LIN {X -0.036,Y -601.709,Z 354.126,A 0.000,B 0.000,C 90.000,E1 238.663} C_DIS
LIN {X -0.086,Y -595.770,Z 354.117,A 0.000,B 0.000,C 90.000,E1 237.089} C_DIS
LIN {X 0.073,Y -585.449,Z 354.101,A 0.000,B 0.000,C 90.000,E1 234.149} C_DIS
LIN {X -0.004,Y -581.907,Z 354.095,A 0.000,B 0.000,C 90.000,E1 233.084} C_DIS
LIN {X -0.070,Y -577.067,Z 354.087,A 0.000,B 0.000,C 90.000,E1 231.743} C_DIS
LIN {X 0.016,Y -567.476,Z 354.072,A 0.000,B 0.000,C 90.000,E1 229.013} C_DIS
LIN {X -0.240,Y -562.093,Z 354.063,A 0.000,B 0.000,C 90.000,E1 227.391} C_DIS
LIN {X -0.222,Y -556.673,Z 354.054,A 0.000,B 0.000,C 90.000,E1 225.729} C_DIS
LIN {X -0.289,Y -550.328,Z 354.043,A 0.000,B 0.000,C 90.000,E1 223.785} C_DIS
LIN {X -0.119,Y -544.951,Z 354.034,A 0.000,B 0.000,C 90.000,E1 222.081} C_DIS
LIN {X -0.053,Y -538.814,Z 354.023,A 0.000,B 0.000,C 90.000,E1 220.092} C_DIS
LIN {X -0.082,Y -532.771,Z 354.012,A 0.000,B 0.000,C 90.000,E1 218.096} C_DIS
LIN {X -0.221,Y -525.363,Z 353.997,A 0.000,B 0.000,C 90.000,E1 215.518} C_DIS
LIN {X 0.006,Y -519.158,Z 353.984,A 0.000,B 0.000,C 90.000,E1 213.166} C_DIS
LIN {X -0.145,Y -512.839,Z 353.970,A 0.000,B 0.000,C 90.000,E1 210.541} C_DIS
LIN {X 0.158,Y -508.202,Z 353.958,A 0.000,B 0.000,C 90.000,E1 208.437} C_DIS
LIN {X 0.158,Y -504.896,Z 353.950,A 0.000,B 0.000,C 90.000,E1 206.950} C_DIS
LIN {X 0.090,Y -501.709,Z 353.942,A 0.000,B 0.000,C 90.000,E1 205.463} C_DIS
LIN {X 0.192,Y -498.425,Z 353.933,A 0.000,B 0.000,C 90.000,E1 203.951} C_DIS
LIN {X 0.088,Y -494.313,Z 353.923,A 0.000,B 0.000,C 90.000,E1 202.153} C_DIS
LIN {X -0.187,Y -491.537,Z 353.916,A 0.000,B 0.000,C 90.000,E1 200.972} C_DIS
LIN {X -0.168,Y -487.311,Z 353.906,A 0.000,B 0.000,C 90.000,E1 199.141} C_DIS
LIN {X -0.098,Y -481.349,Z 353.891,A 0.000,B 0.000,C 90.000,E1 196.370} C_DIS
LIN {X 0.032,Y -476.989,Z 353.879,A 0.000,B 0.000,C 90.000,E1 194.189} C_DIS
LIN {X 0.059,Y -472.858,Z 353.867,A 0.000,B 0.000,C 90.000,E1 192.007} C_DIS
LIN {X -0.222,Y -468.764,Z 353.855,A 0.000,B 0.000,C 90.000,E1 189.849} C_DIS
LIN {X -0.227,Y -465.034,Z 353.842,A 0.000,B 0.000,C 90.000,E1 187.644} C_DIS
LIN {X -0.207,Y -461.052,Z 353.828,A 0.000,B 0.000,C 90.000,E1 185.106} C_DIS
LIN {X 0.195,Y -456.557,Z 353.809,A 0.000,B 0.000,C 90.000,E1 181.547} C_DIS
LIN {X -0.196,Y -452.824,Z 353.786,A 0.000,B 0.000,C 90.000,E1 177.421} C_DIS
LIN {X 0.187,Y -451.196,Z 353.768,A 0.000,B 0.000,C 90.000,E1 174.147} C_DIS
LIN {X 0.099,Y -450.799,Z 353.743,A 0.000,B 0.000,C 90.000,E1 169.634} C_DIS
LIN {X -0.141,Y -451.606,Z 353.726,A 0.000,B 0.000,C 90.000,E1 166.756} C_DIS
LIN {X 0.146,Y -454.119,Z 353.705,A 0.000,B 0.000,C 90.000,E1 162.851} C_DIS
LIN {X -0.169,Y -458.577,Z 353.682,A 0.000,B 0.000,C 90.000,E1 158.720} C_DIS
LIN {X 0.269,Y -464.355,Z 353.660,A 0.000,B 0.000,C 90.000,E1 154.845} C_DIS
LIN {X -0.128,Y -472.523,Z 353.638,A 0.000,B 0.000,C 90.000,E1 150.795} C_DIS
LIN {X 0.032,Y -482.123,Z 353.617,A 0.000,B 0.000,C 90.000,E1 147.041} C_DIS
LIN {X 0.035,Y -490.562,Z 353.602,A 0.000,B 0.000,C 90.000,E1 144.276} C_DIS
LIN {X -0.182,Y -496.597,Z 353.591,A 0.000,B 0.000,C 90.000,E1 142.477} C_DIS
LIN {X 0.047,Y -502.541,Z 353.581,A 0.000,B 0.000,C 90.000,E1 140.642} C_DIS
LIN {X -0.094,Y -506.324,Z 353.575,A 0.000,B 0.000,C 90.000,E1 139.461} C_DIS
LIN {X 0.147,Y -509.852,Z 353.568,A 0.000,B 0.000,C 90.000,E1 138.243} C_DIS
LIN {X -0.188,Y -512.384,Z 353.563,A 0.000,B 0.000,C 90.000,E1 137.391} C_DIS
LIN {X -0.238,Y -515.302,Z 353.557,A 0.000,B 0.000,C 90.000,E1 136.215} C_DIS
LIN {X 0.298,Y -516.581,Z 353.553,A 0.000,B 0.000,C 90.000,E1 135.567} C_DIS
LIN {X 0.024,Y -518.323,Z 353.548,A 0.000,B 0.000,C 90.000,E1 134.717} C_DIS
LIN {X 0.222,Y -519.271,Z 353.545,A 0.000,B 0.000,C 90.000,E1 134.109} C_DIS
LIN {X -0.014,Y -520.436,Z 353.540,A 0.000,B 0.000,C 90.000,E1 133.257} C_DIS
LIN {X 0.056,Y -521.438,Z 353.534,A 0.000,B 0.000,C 90.000,E1 132.081} C_DIS
LIN {X -0.154,Y -521.848,Z 353.529,A 0.000,B 0.000,C 90.000,E1 131.229} C_DIS
LIN {X 0.318,Y -521.762,Z 353.523,A 0.000,B 0.000,C 90.000,E1 130.011} C_DIS
LIN {X -0.233,Y -521.317,Z 353.518,A 0.000,B 0.000,C 90.000,E1 129.197} C_DIS
LIN {X -0.055,Y -520.533,Z 353.513,A 0.000,B 0.000,C 90.000,E1 128.302} C_DIS
LIN {X -0.209,Y -519.480,Z 353.508,A 0.000,B 0.000,C 90.000,E1 127.443} C_DIS
LIN {X -0.069,Y -517.552,Z 353.500,A 0.000,B 0.000,C 90.000,E1 125.964} C_DIS
LIN {X -0.253,Y -516.241,Z 353.495,A 0.000,B 0.000,C 90.000,E1 125.105} C_DIS
LIN {X -0.030,Y -514.817,Z 353.490,A 0.000,B 0.000,C 90.000,E1 124.199} C_DIS
LIN {X 0.092,Y -512.635,Z 353.483,A 0.000,B 0.000,C 90.000,E1 123.007} C_DIS
LIN {X -0.013,Y -510.853,Z 353.479,A 0.000,B 0.000,C 90.000,E1 122.133} C_DIS
LIN {X 0.199,Y -508.213,Z 353.472,A 0.000,B 0.000,C 90.000,E1 120.924} C_DIS
LIN {X 0.114,Y -505.440,Z 353.465,A 0.000,B 0.000,C 90.000,E1 119.745} C_DIS
LIN {X -0.005,Y -502.430,Z 353.459,A 0.000,B 0.000,C 90.000,E1 118.565} C_DIS
LIN {X -0.114,Y -498.474,Z 353.450,A 0.000,B 0.000,C 90.000,E1 117.078} C_DIS
LIN {X 0.146,Y -494.271,Z 353.442,A 0.000,B 0.000,C 90.000,E1 115.540} C_DIS
LIN {X 0.037,Y -491.575,Z 353.437,A 0.000,B 0.000,C 90.000,E1 114.643} C_DIS
LIN {X -0.058,Y -486.521,Z 353.429,A 0.000,B 0.000,C 90.000,E1 113.131} C_DIS
LIN {X 0.001,Y -482.302,Z 353.422,A 0.000,B 0.000,C 90.000,E1 111.897} C_DIS
LIN {X 0.004,Y -478.925,Z 353.417,A 0.000,B 0.000,C 90.000,E1 110.972} C_DIS
LIN {X 0.197,Y -475.980,Z 353.412,A 0.000,B 0.000,C 90.000,E1 110.174} C_DIS
LIN {X 0.128,Y -470.325,Z 353.404,A 0.000,B 0.000,C 90.000,E1 108.779} C_DIS
LIN {X 0.209,Y -465.075,Z 353.397,A 0.000,B 0.000,C 90.000,E1 107.511} C_DIS
LIN {X -0.253,Y -462.804,Z 353.395,A 0.000,B 0.000,C 90.000,E1 107.040} C_DIS
LIN {X 0.150,Y -462.797,Z 353.395,A 0.000,B 0.000,C 90.000,E1 106.985} C_DIS
LIN {X -0.040,Y -467.514,Z 353.383,A 0.000,B 0.000,C 90.000,E1 105.009} C_DIS
LIN {X -0.235,Y -468.097,Z 353.382,A 0.000,B 0.000,C 90.000,E1 104.717} C_DIS
LIN {X -0.096,Y -475.756,Z 353.357,A 0.000,B 0.000,C 90.000,E1 100.310} C_DIS
LIN {X 0.210,Y -476.285,Z 353.356,A 0.000,B 0.000,C 90.000,E1 99.962} C_DIS
LIN {X 0.158,Y -481.755,Z 353.331,A 0.000,B 0.000,C 90.000,E1 95.625} C_DIS
LIN {X 0.005,Y -482.163,Z 353.330,A 0.000,B 0.000,C 90.000,E1 95.334} C_DIS
LIN {X -0.066,Y -485.285,Z 353.306,A 0.000,B 0.000,C 90.000,E1 91.031} C_DIS
LIN {X -0.241,Y -485.538,Z 353.304,A 0.000,B 0.000,C 90.000,E1 90.745} C_DIS
LIN {X -0.034,Y -486.309,Z 353.282,A 0.000,B 0.000,C 90.000,E1 86.731} C_DIS
LIN {X 0.101,Y -486.319,Z 353.278,A 0.000,B 0.000,C 90.000,E1 86.102} C_DIS
LIN {X 0.174,Y -484.623,Z 353.253,A 0.000,B 0.000,C 90.000,E1 81.489} C_DIS
LIN {X 0.054,Y -480.552,Z 353.227,A 0.000,B 0.000,C 90.000,E1 76.881} C_DIS
LIN {X 0.150,Y -476.599,Z 353.212,A 0.000,B 0.000,C 90.000,E1 74.212} C_DIS
LIN {X 0.109,Y -476.610,Z 353.212,A 0.000,B 0.000,C 90.000,E1 74.212} C_DIS
LIN {X -0.055,Y -479.016,Z 353.210,A 0.000,B 0.000,C 90.000,E1 73.795} C_DIS
LIN {X 0.227,Y -482.346,Z 353.207,A 0.000,B 0.000,C 90.000,E1 73.142} C_DIS
LIN {X -0.158,Y -484.629,Z 353.204,A 0.000,B 0.000,C 90.000,E1 72.725} C_DIS
LIN {X -0.159,Y -486.303,Z 353.202,A 0.000,B 0.000,C 90.000,E1 72.417} C_DIS
LIN {X -0.046,Y -490.120,Z 353.198,A 0.000,B 0.000,C 90.000,E1 71.638} C_DIS
LIN {X 0.102,Y -493.632,Z 353.194,A 0.000,B 0.000,C 90.000,E1 70.859} C_DIS
LIN {X 0.240,Y -497.512,Z 353.189,A 0.000,B 0.000,C 90.000,E1 69.934} C_DIS
LIN {X -0.019,Y -500.472,Z 353.185,A 0.000,B 0.000,C 90.000,E1 69.209} C_DIS
LIN {X 0.195,Y -503.659,Z 353.180,A 0.000,B 0.000,C 90.000,E1 68.284} C_DIS
LIN {X -0.108,Y -505.682,Z 353.176,A 0.000,B 0.000,C 90.000,E1 67.720} C_DIS
LIN {X 0.267,Y -509.497,Z 353.170,A 0.000,B 0.000,C 90.000,E1 66.485} C_DIS
LIN {X -0.242,Y -513.111,Z 353.163,A 0.000,B 0.000,C 90.000,E1 65.357} C_DIS
LIN {X -0.020,Y -516.555,Z 353.156,A 0.000,B 0.000,C 90.000,E1 64.152} C_DIS
LIN {X -0.210,Y -519.929,Z 353.150,A 0.000,B 0.000,C 90.000,E1 62.999} C_DIS
LIN {X 0.031,Y -523.998,Z 353.142,A 0.000,B 0.000,C 90.000,E1 61.513} C_DIS
LIN {X -0.165,Y -528.825,Z 353.132,A 0.000,B 0.000,C 90.000,E1 59.793} C_DIS
LIN {X 0.065,Y -532.061,Z 353.126,A 0.000,B 0.000,C 90.000,E1 58.614} C_DIS
LIN {X 0.156,Y -536.027,Z 353.118,A 0.000,B 0.000,C 90.000,E1 57.168} C_DIS
LIN {X -0.137,Y -538.289,Z 353.113,A 0.000,B 0.000,C 90.000,E1 56.342} C_DIS
LIN {X 0.055,Y -541.226,Z 353.107,A 0.000,B 0.000,C 90.000,E1 55.182} C_DIS
LIN {X 0.126,Y -543.291,Z 353.102,A 0.000,B 0.000,C 90.000,E1 54.322} C_DIS
LIN {X -0.064,Y -545.864,Z 353.096,A 0.000,B 0.000,C 90.000,E1 53.210} C_DIS
LIN {X 0.101,Y -548.220,Z 353.089,A 0.000,B 0.000,C 90.000,E1 52.065} C_DIS
LIN {X -0.135,Y -550.313,Z 353.083,A 0.000,B 0.000,C 90.000,E1 50.964} C_DIS
LIN {X -0.046,Y -551.569,Z 353.078,A 0.000,B 0.000,C 90.000,E1 50.114} C_DIS
LIN {X 0.124,Y -552.673,Z 353.074,A 0.000,B 0.000,C 90.000,E1 49.256} C_DIS
LIN {X 0.187,Y -553.299,Z 353.071,A 0.000,B 0.000,C 90.000,E1 48.690} C_DIS
LIN {X -0.053,Y -553.923,Z 353.066,A 0.000,B 0.000,C 90.000,E1 47.877} C_DIS
LIN {X 0.110,Y -554.260,Z 353.060,A 0.000,B 0.000,C 90.000,E1 46.743} C_DIS
LIN {X -0.099,Y -553.911,Z 353.054,A 0.000,B 0.000,C 90.000,E1 45.648} C_DIS
LIN {X -0.013,Y -553.795,Z 353.051,A 0.000,B 0.000,C 90.000,E1 45.081} C_DIS
LIN {X -0.277,Y -553.292,Z 353.046,A 0.000,B 0.000,C 90.000,E1 44.271} C_DIS
LIN {X 0.232,Y -552.603,Z 353.041,A 0.000,B 0.000,C 90.000,E1 43.380} C_DIS
LIN {X 0.353,Y -551.766,Z 353.037,A 0.000,B 0.000,C 90.000,E1 42.528} C_DIS
LIN {X 0.103,Y -550.394,Z 353.030,A 0.000,B 0.000,C 90.000,E1 41.434} C_DIS
LIN {X -0.111,Y -549.020,Z 353.024,A 0.000,B 0.000,C 90.000,E1 40.334} C_DIS
LIN {X 0.106,Y -546.765,Z 353.015,A 0.000,B 0.000,C 90.000,E1 38.624} C_DIS
LIN {X -0.034,Y -544.148,Z 353.004,A 0.000,B 0.000,C 90.000,E1 36.664} C_DIS
LIN {X -0.125,Y -541.563,Z 352.993,A 0.000,B 0.000,C 90.000,E1 34.692} C_DIS
LIN {X 0.143,Y -539.420,Z 352.983,A 0.000,B 0.000,C 90.000,E1 32.959} C_DIS
LIN {X 0.063,Y -537.711,Z 352.975,A 0.000,B 0.000,C 90.000,E1 31.544} C_DIS
LIN {X 0.120,Y -535.461,Z 352.964,A 0.000,B 0.000,C 90.000,E1 29.539} C_DIS
LIN {X -0.121,Y -533.665,Z 352.955,A 0.000,B 0.000,C 90.000,E1 27.847} C_DIS
LIN {X 0.070,Y -531.827,Z 352.945,A 0.000,B 0.000,C 90.000,E1 26.104} C_DIS
LIN {X -0.020,Y -530.149,Z 352.936,A 0.000,B 0.000,C 90.000,E1 24.387} C_DIS
LIN {X -0.009,Y -528.086,Z 352.923,A 0.000,B 0.000,C 90.000,E1 22.078} C_DIS
LIN {X -0.119,Y -526.755,Z 352.913,A 0.000,B 0.000,C 90.000,E1 20.355} C_DIS
LIN {X 0.054,Y -525.512,Z 352.902,A 0.000,B 0.000,C 90.000,E1 18.308} C_DIS
LIN {X -0.135,Y -524.223,Z 352.886,A 0.000,B 0.000,C 90.000,E1 15.426} C_DIS
LIN {X 0.207,Y -523.658,Z 352.873,A 0.000,B 0.000,C 90.000,E1 13.063} C_DIS
LIN {X -0.178,Y -523.669,Z 352.857,A 0.000,B 0.000,C 90.000,E1 10.197} C_DIS
LIN {X -0.237,Y -524.304,Z 352.842,A 0.000,B 0.000,C 90.000,E1 7.587} C_DIS
LIN {X 0.156,Y -525.263,Z 352.831,A 0.000,B 0.000,C 90.000,E1 5.511} C_DIS
LIN {X -0.098,Y -527.568,Z 352.813,A 0.000,B 0.000,C 90.000,E1 2.350} C_DIS
LIN {X 0.124,Y -532.150,Z 352.791,A 0.000,B 0.000,C 90.000,E1 358.339} C_DIS
LIN {X 0.135,Y -536.021,Z 352.777,A 0.000,B 0.000,C 90.000,E1 355.755} C_DIS
LIN {X 0.214,Y -538.991,Z 352.767,A 0.000,B 0.000,C 90.000,E1 354.033} C_DIS
LIN {X -0.103,Y -546.936,Z 352.745,A 0.000,B 0.000,C 90.000,E1 350.095} C_DIS
LIN {X -0.130,Y -557.070,Z 352.723,A 0.000,B 0.000,C 90.000,E1 346.172} C_DIS
LIN {X -0.249,Y -561.959,Z 352.714,A 0.000,B 0.000,C 90.000,E1 344.519} C_DIS
LIN {X 0.204,Y -567.954,Z 352.703,A 0.000,B 0.000,C 90.000,E1 342.543} C_DIS
LIN {X 0.118,Y -571.423,Z 352.697,A 0.000,B 0.000,C 90.000,E1 341.456} C_DIS
LIN {X -0.091,Y -577.549,Z 352.686,A 0.000,B 0.000,C 90.000,E1 339.571} C_DIS
LIN {X -0.207,Y -581.837,Z 352.679,A 0.000,B 0.000,C 90.000,E1 338.230} C_DIS
LIN {X -0.038,Y -586.185,Z 352.672,A 0.000,B 0.000,C 90.000,E1 336.869} C_DIS
LIN {X 0.232,Y -592.388,Z 352.661,A 0.000,B 0.000,C 90.000,E1 334.973} C_DIS
LIN {X 0.126,Y -598.741,Z 352.651,A 0.000,B 0.000,C 90.000,E1 333.127} C_DIS
LIN {X -0.152,Y -606.023,Z 352.639,A 0.000,B 0.000,C 90.000,E1 331.051} C_DIS
LIN {X 0.098,Y -612.474,Z 352.629,A 0.000,B 0.000,C 90.000,E1 329.203} C_DIS
LIN {X 0.027,Y -617.167,Z 352.622,A 0.000,B 0.000,C 90.000,E1 327.916} C_DIS
LIN {X -0.179,Y -623.539,Z 352.612,A 0.000,B 0.000,C 90.000,E1 326.135} C_DIS
LIN {X -0.060,Y -627.038,Z 352.606,A 0.000,B 0.000,C 90.000,E1 325.102} C_DIS
LIN {X 0.100,Y -630.523,Z 352.600,A 0.000,B 0.000,C 90.000,E1 324.069} C_DIS
LIN {X -0.348,Y -634.734,Z 352.593,A 0.000,B 0.000,C 90.000,E1 322.844} C_DIS
LIN {X -0.220,Y -638.066,Z 352.588,A 0.000,B 0.000,C 90.000,E1 321.823} C_DIS
LIN {X 0.082,Y -645.573,Z 352.575,A 0.000,B 0.000,C 90.000,E1 319.542} C_DIS
LIN {X 0.349,Y -648.065,Z 352.571,A 0.000,B 0.000,C 90.000,E1 318.771} C_DIS
LIN {X -0.047,Y -654.556,Z 352.560,A 0.000,B 0.000,C 90.000,E1 316.824} C_DIS
LIN {X 0.251,Y -658.820,Z 352.553,A 0.000,B 0.000,C 90.000,E1 315.567} C_DIS
LIN {X 0.144,Y -662.808,Z 352.547,A 0.000,B 0.000,C 90.000,E1 314.352} C_DIS
LIN {X 0.095,Y -666.849,Z 352.540,A 0.000,B 0.000,C 90.000,E1 313.137} C_DIS
LIN {X 0.143,Y -670.838,Z 352.533,A 0.000,B 0.000,C 90.000,E1 311.919} C_DIS
LIN {X -0.273,Y -673.068,Z 352.529,A 0.000,B 0.000,C 90.000,E1 311.229} C_DIS
LIN {X -0.103,Y -677.383,Z 352.521,A 0.000,B 0.000,C 90.000,E1 309.769} C_DIS
LIN {X -0.348,Y -680.155,Z 352.516,A 0.000,B 0.000,C 90.000,E1 308.830} C_DIS
LIN {X -0.160,Y -682.135,Z 352.512,A 0.000,B 0.000,C 90.000,E1 308.096} C_DIS
LIN {X 0.047,Y -684.030,Z 352.508,A 0.000,B 0.000,C 90.000,E1 307.363} C_DIS
LIN {X -0.142,Y -685.745,Z 352.504,A 0.000,B 0.000,C 90.000,E1 306.664} C_DIS
LIN {X 0.095,Y -687.302,Z 352.500,A 0.000,B 0.000,C 90.000,E1 305.931} C_DIS
LIN {X -0.061,Y -688.724,Z 352.496,A 0.000,B 0.000,C 90.000,E1 305.231} C_DIS
LIN {X 0.004,Y -690.340,Z 352.490,A 0.000,B 0.000,C 90.000,E1 304.278} C_DIS
LIN {X 0.240,Y -691.079,Z 352.488,A 0.000,B 0.000,C 90.000,E1 303.785} C_DIS
LIN {X 0.120,Y -691.887,Z 352.484,A 0.000,B 0.000,C 90.000,E1 303.086} C_DIS
LIN {X -0.370,Y -692.452,Z 352.480,A 0.000,B 0.000,C 90.000,E1 302.418} C_DIS
LIN {X -0.129,Y -692.749,Z 352.477,A 0.000,B 0.000,C 90.000,E1 301.926} C_DIS
LIN {X -0.018,Y -692.924,Z 352.473,A 0.000,B 0.000,C 90.000,E1 301.209} C_DIS
LIN {X -0.141,Y -692.709,Z 352.469,A 0.000,B 0.000,C 90.000,E1 300.512} C_DIS
LIN {X 0.336,Y -692.443,Z 352.467,A 0.000,B 0.000,C 90.000,E1 300.001} C_DIS
LIN {X -0.149,Y -691.768,Z 352.463,A 0.000,B 0.000,C 90.000,E1 299.333} C_DIS
LIN {X 0.330,Y -691.250,Z 352.460,A 0.000,B 0.000,C 90.000,E1 298.821} C_DIS
LIN {X 0.200,Y -690.536,Z 352.458,A 0.000,B 0.000,C 90.000,E1 298.359} C_DIS
LIN {X -0.161,Y -688.395,Z 352.451,A 0.000,B 0.000,C 90.000,E1 297.206} C_DIS
LIN {X 0.145,Y -686.482,Z 352.446,A 0.000,B 0.000,C 90.000,E1 296.232} C_DIS
LIN {X 0.119,Y -684.425,Z 352.441,A 0.000,B 0.000,C 90.000,E1 295.283} C_DIS
LIN {X 0.275,Y -681.593,Z 352.434,A 0.000,B 0.000,C 90.000,E1 294.079} C_DIS
LIN {X 0.108,Y -678.643,Z 352.427,A 0.000,B 0.000,C 90.000,E1 292.898} C_DIS
LIN {X 0.070,Y -674.903,Z 352.419,A 0.000,B 0.000,C 90.000,E1 291.461} C_DIS
LIN {X 0.331,Y -671.189,Z 352.411,A 0.000,B 0.000,C 90.000,E1 289.993} C_DIS
LIN {X 0.340,Y -666.277,Z 352.401,A 0.000,B 0.000,C 90.000,E1 288.055} C_DIS
LIN {X -0.078,Y -661.151,Z 352.388,A 0.000,B 0.000,C 90.000,E1 285.898} C_DIS
LIN {X 0.338,Y -655.982,Z 352.375,A 0.000,B 0.000,C 90.000,E1 283.411} C_DIS
LIN {X 0.287,Y -650.238,Z 352.356,A 0.000,B 0.000,C 90.000,E1 279.962} C_DIS
LIN {X -0.175,Y -646.632,Z 352.338,A 0.000,B 0.000,C 90.000,E1 276.777} C_DIS
LIN {X 0.307,Y -644.934,Z 352.324,A 0.000,B 0.000,C 90.000,E1 274.245} C_DIS
LIN {X -0.195,Y -643.928,Z 352.309,A 0.000,B 0.000,C 90.000,E1 271.547} C_DIS
LIN {X 0.039,Y -643.973,Z 352.291,A 0.000,B 0.000,C 90.000,E1 268.282} C_DIS
LIN {X -0.053,Y -644.813,Z 352.278,A 0.000,B 0.000,C 90.000,E1 266.045} C_DIS
LIN {X -0.248,Y -645.674,Z 352.268,A 0.000,B 0.000,C 90.000,E1 264.318} C_DIS
LIN {X 0.060,Y -646.746,Z 352.257,A 0.000,B 0.000,C 90.000,E1 262.299} C_DIS
LIN {X 0.235,Y -647.709,Z 352.249,A 0.000,B 0.000,C 90.000,E1 260.792} C_DIS
LIN {X -0.214,Y -648.417,Z 352.241,A 0.000,B 0.000,C 90.000,E1 259.342} C_DIS
LIN {X -0.038,Y -649.497,Z 352.231,A 0.000,B 0.000,C 90.000,E1 257.589} C_DIS
LIN {X -0.069,Y -650.286,Z 352.224,A 0.000,B 0.000,C 90.000,E1 256.353} C_DIS
LIN {X 0.040,Y -650.605,Z 352.219,A 0.000,B 0.000,C 90.000,E1 255.353} C_DIS
LIN {X -0.180,Y -650.543,Z 352.215,A 0.000,B 0.000,C 90.000,E1 254.629} C_DIS
LIN {X 0.055,Y -650.235,Z 352.210,A 0.000,B 0.000,C 90.000,E1 253.866} C_DIS
LIN {X -0.026,Y -649.906,Z 352.208,A 0.000,B 0.000,C 90.000,E1 253.378} C_DIS
LIN {X -0.293,Y -649.419,Z 352.205,A 0.000,B 0.000,C 90.000,E1 252.906} C_DIS
LIN {X 0.107,Y -648.522,Z 352.201,A 0.000,B 0.000,C 90.000,E1 252.127} C_DIS
LIN {X -0.119,Y -647.394,Z 352.197,A 0.000,B 0.000,C 90.000,E1 251.402} C_DIS
LIN {X -0.142,Y -645.989,Z 352.193,A 0.000,B 0.000,C 90.000,E1 250.659} C_DIS
LIN {X 0.218,Y -644.275,Z 352.188,A 0.000,B 0.000,C 90.000,E1 249.880} C_DIS
LIN {X -0.055,Y -642.261,Z 352.184,A 0.000,B 0.000,C 90.000,E1 249.156} C_DIS
LIN {X -0.117,Y -640.053,Z 352.180,A 0.000,B 0.000,C 90.000,E1 248.411} C_DIS
LIN {X -0.197,Y -637.645,Z 352.176,A 0.000,B 0.000,C 90.000,E1 247.667} C_DIS
LIN {X -0.300,Y -634.951,Z 352.172,A 0.000,B 0.000,C 90.000,E1 246.922} C_DIS
LIN {X 0.214,Y -630.362,Z 352.165,A 0.000,B 0.000,C 90.000,E1 245.613} C_DIS
LIN {X 0.318,Y -626.508,Z 352.159,A 0.000,B 0.000,C 90.000,E1 244.588} C_DIS
LIN {X 0.105,Y -621.473,Z 352.152,A 0.000,B 0.000,C 90.000,E1 243.332} C_DIS
LIN {X 0.364,Y -616.434,Z 352.145,A 0.000,B 0.000,C 90.000,E1 242.025} C_DIS
LIN {X -0.289,Y -611.398,Z 352.138,A 0.000,B 0.000,C 90.000,E1 240.795} C_DIS
LIN {X -0.008,Y -604.242,Z 352.128,A 0.000,B 0.000,C 90.000,E1 238.948} C_DIS
LIN {X -0.106,Y -597.338,Z 352.117,A 0.000,B 0.000,C 90.000,E1 237.120} C_DIS
LIN {X 0.152,Y -586.075,Z 352.100,A 0.000,B 0.000,C 90.000,E1 233.909} C_DIS
LIN {X 0.089,Y -582.466,Z 352.094,A 0.000,B 0.000,C 90.000,E1 232.844} C_DIS
LIN {X -0.317,Y -577.576,Z 352.086,A 0.000,B 0.000,C 90.000,E1 231.537} C_DIS
LIN {X 0.154,Y -568.071,Z 352.071,A 0.000,B 0.000,C 90.000,E1 228.771} C_DIS
LIN {X -0.086,Y -562.724,Z 352.062,A 0.000,B 0.000,C 90.000,E1 227.148} C_DIS
LIN {X -0.056,Y -557.280,Z 352.053,A 0.000,B 0.000,C 90.000,E1 225.486} C_DIS
LIN {X -0.110,Y -550.961,Z 352.042,A 0.000,B 0.000,C 90.000,E1 223.542} C_DIS
LIN {X 0.070,Y -545.560,Z 352.033,A 0.000,B 0.000,C 90.000,E1 221.838} C_DIS
LIN {X -0.223,Y -540.315,Z 352.023,A 0.000,B 0.000,C 90.000,E1 220.172} C_DIS
LIN {X -0.208,Y -533.404,Z 352.010,A 0.000,B 0.000,C 90.000,E1 217.890} C_DIS
LIN {X -0.296,Y -526.817,Z 351.998,A 0.000,B 0.000,C 90.000,E1 215.598} C_DIS
LIN {X -0.020,Y -520.568,Z 351.985,A 0.000,B 0.000,C 90.000,E1 213.245} C_DIS
LIN {X -0.204,Y -513.563,Z 351.968,A 0.000,B 0.000,C 90.000,E1 210.335} C_DIS
LIN {X 0.115,Y -508.957,Z 351.957,A 0.000,B 0.000,C 90.000,E1 208.231} C_DIS
LIN {X 0.063,Y -504.400,Z 351.945,A 0.000,B 0.000,C 90.000,E1 206.155} C_DIS
LIN {X 0.213,Y -501.191,Z 351.937,A 0.000,B 0.000,C 90.000,E1 204.643} C_DIS
LIN {X -0.029,Y -499.181,Z 351.932,A 0.000,B 0.000,C 90.000,E1 203.770} C_DIS
LIN {X -0.111,Y -495.103,Z 351.922,A 0.000,B 0.000,C 90.000,E1 201.972} C_DIS
LIN {X 0.131,Y -491.635,Z 351.914,A 0.000,B 0.000,C 90.000,E1 200.429} C_DIS
LIN {X 0.017,Y -486.748,Z 351.902,A 0.000,B 0.000,C 90.000,E1 198.308} C_DIS
LIN {X 0.086,Y -481.589,Z 351.888,A 0.000,B 0.000,C 90.000,E1 195.843} C_DIS
LIN {X -0.118,Y -477.269,Z 351.876,A 0.000,B 0.000,C 90.000,E1 193.703} C_DIS
LIN {X 0.127,Y -474.364,Z 351.867,A 0.000,B 0.000,C 90.000,E1 192.119} C_DIS
LIN {X -0.122,Y -470.271,Z 351.855,A 0.000,B 0.000,C 90.000,E1 189.962} C_DIS
LIN {X -0.093,Y -466.509,Z 351.843,A 0.000,B 0.000,C 90.000,E1 187.757} C_DIS
LIN {X -0.034,Y -462.509,Z 351.829,A 0.000,B 0.000,C 90.000,E1 185.220} C_DIS
LIN {X 0.157,Y -457.585,Z 351.808,A 0.000,B 0.000,C 90.000,E1 181.375} C_DIS
LIN {X -0.182,Y -453.881,Z 351.785,A 0.000,B 0.000,C 90.000,E1 177.249} C_DIS
LIN {X -0.211,Y -452.303,Z 351.767,A 0.000,B 0.000,C 90.000,E1 174.033} C_DIS
LIN {X 0.075,Y -451.932,Z 351.743,A 0.000,B 0.000,C 90.000,E1 169.803} C_DIS
LIN {X 0.165,Y -452.438,Z 351.731,A 0.000,B 0.000,C 90.000,E1 167.533} C_DIS
LIN {X 0.005,Y -455.354,Z 351.704,A 0.000,B 0.000,C 90.000,E1 162.725} C_DIS
LIN {X 0.103,Y -460.240,Z 351.679,A 0.000,B 0.000,C 90.000,E1 158.230} C_DIS
LIN {X 0.259,Y -465.592,Z 351.660,A 0.000,B 0.000,C 90.000,E1 154.717} C_DIS
LIN {X 0.116,Y -471.078,Z 351.644,A 0.000,B 0.000,C 90.000,E1 151.897} C_DIS
LIN {X -0.081,Y -480.873,Z 351.621,A 0.000,B 0.000,C 90.000,E1 147.867} C_DIS
LIN {X -0.054,Y -490.940,Z 351.603,A 0.000,B 0.000,C 90.000,E1 144.482} C_DIS
LIN {X -0.006,Y -497.960,Z 351.591,A 0.000,B 0.000,C 90.000,E1 142.351} C_DIS
LIN {X -0.142,Y -503.805,Z 351.581,A 0.000,B 0.000,C 90.000,E1 140.561} C_DIS
LIN {X -0.264,Y -507.497,Z 351.574,A 0.000,B 0.000,C 90.000,E1 139.380} C_DIS
LIN {X -0.006,Y -510.988,Z 351.568,A 0.000,B 0.000,C 90.000,E1 138.162} C_DIS
LIN {X 0.048,Y -513.408,Z 351.563,A 0.000,B 0.000,C 90.000,E1 137.268} C_DIS
LIN {X 0.099,Y -515.508,Z 351.558,A 0.000,B 0.000,C 90.000,E1 136.377} C_DIS
LIN {X -0.094,Y -516.782,Z 351.555,A 0.000,B 0.000,C 90.000,E1 135.810} C_DIS
LIN {X 0.001,Y -518.448,Z 351.550,A 0.000,B 0.000,C 90.000,E1 134.919} C_DIS
LIN {X 0.116,Y -519.762,Z 351.545,A 0.000,B 0.000,C 90.000,E1 134.028} C_DIS
LIN {X -0.047,Y -520.329,Z 351.541,A 0.000,B 0.000,C 90.000,E1 133.461} C_DIS
LIN {X -0.116,Y -520.739,Z 351.540,A 0.000,B 0.000,C 90.000,E1 133.176} C_DIS
LIN {X -0.043,Y -521.472,Z 351.533,A 0.000,B 0.000,C 90.000,E1 132.000} C_DIS
LIN {X -0.254,Y -521.802,Z 351.529,A 0.000,B 0.000,C 90.000,E1 131.148} C_DIS
LIN {X -0.070,Y -521.676,Z 351.524,A 0.000,B 0.000,C 90.000,E1 130.253} C_DIS
LIN {X 0.116,Y -521.274,Z 351.519,A 0.000,B 0.000,C 90.000,E1 129.358} C_DIS
LIN {X 0.294,Y -520.500,Z 351.514,A 0.000,B 0.000,C 90.000,E1 128.463} C_DIS
LIN {X 0.140,Y -519.453,Z 351.509,A 0.000,B 0.000,C 90.000,E1 127.604} C_DIS
LIN {X -0.135,Y -517.505,Z 351.501,A 0.000,B 0.000,C 90.000,E1 126.171} C_DIS
LIN {X 0.038,Y -515.715,Z 351.494,A 0.000,B 0.000,C 90.000,E1 124.978} C_DIS
LIN {X 0.182,Y -513.742,Z 351.488,A 0.000,B 0.000,C 90.000,E1 123.785} C_DIS
LIN {X 0.008,Y -511.499,Z 351.481,A 0.000,B 0.000,C 90.000,E1 122.625} C_DIS
LIN {X -0.199,Y -509.000,Z 351.475,A 0.000,B 0.000,C 90.000,E1 121.465} C_DIS
LIN {X -0.015,Y -506.324,Z 351.468,A 0.000,B 0.000,C 90.000,E1 120.256} C_DIS
LIN {X 0.181,Y -502.690,Z 351.460,A 0.000,B 0.000,C 90.000,E1 118.743} C_DIS
LIN {X 0.069,Y -498.798,Z 351.452,A 0.000,B 0.000,C 90.000,E1 117.257} C_DIS
LIN {X 0.012,Y -496.374,Z 351.447,A 0.000,B 0.000,C 90.000,E1 116.360} C_DIS
LIN {X -0.027,Y -493.007,Z 351.440,A 0.000,B 0.000,C 90.000,E1 115.155} C_DIS
LIN {X 0.259,Y -491.242,Z 351.436,A 0.000,B 0.000,C 90.000,E1 114.515} C_DIS
LIN {X -0.037,Y -486.390,Z 351.428,A 0.000,B 0.000,C 90.000,E1 113.025} C_DIS
LIN {X 0.211,Y -481.312,Z 351.419,A 0.000,B 0.000,C 90.000,E1 111.461} C_DIS
LIN {X 0.021,Y -476.835,Z 351.413,A 0.000,B 0.000,C 90.000,E1 110.248} C_DIS
LIN {X 0.166,Y -472.653,Z 351.406,A 0.000,B 0.000,C 90.000,E1 109.141} C_DIS
LIN {X -0.105,Y -467.033,Z 351.399,A 0.000,B 0.000,C 90.000,E1 107.764} C_DIS
LIN {X -0.197,Y -463.197,Z 351.394,A 0.000,B 0.000,C 90.000,E1 106.858} C_DIS
LIN {X -0.237,Y -463.181,Z 351.394,A 0.000,B 0.000,C 90.000,E1 106.858} C_DIS
LIN {X 0.054,Y -467.757,Z 351.383,A 0.000,B 0.000,C 90.000,E1 104.898} C_DIS
LIN {X 0.027,Y -475.963,Z 351.357,A 0.000,B 0.000,C 90.000,E1 100.197} C_DIS
LIN {X 0.175,Y -476.676,Z 351.353,A 0.000,B 0.000,C 90.000,E1 99.557} C_DIS
LIN {X -0.179,Y -481.911,Z 351.331,A 0.000,B 0.000,C 90.000,E1 95.568} C_DIS
LIN {X 0.149,Y -482.202,Z 351.329,A 0.000,B 0.000,C 90.000,E1 95.220} C_DIS
LIN {X 0.087,Y -485.389,Z 351.305,A 0.000,B 0.000,C 90.000,E1 90.917} C_DIS
LIN {X -0.089,Y -485.529,Z 351.303,A 0.000,B 0.000,C 90.000,E1 90.630} C_DIS
LIN {X 0.120,Y -486.357,Z 351.281,A 0.000,B 0.000,C 90.000,E1 86.617} C_DIS
LIN {X -0.056,Y -486.369,Z 351.280,A 0.000,B 0.000,C 90.000,E1 86.331} C_DIS
LIN {X -0.066,Y -485.859,Z 351.275,A 0.000,B 0.000,C 90.000,E1 85.412} C_DIS
LIN {X -0.033,Y -484.692,Z 351.254,A 0.000,B 0.000,C 90.000,E1 81.724} C_DIS
LIN {X -0.164,Y -484.507,Z 351.252,A 0.000,B 0.000,C 90.000,E1 81.432} C_DIS
LIN {X 0.174,Y -480.441,Z 351.227,A 0.000,B 0.000,C 90.000,E1 76.769} C_DIS
LIN {X 0.067,Y -476.750,Z 351.213,A 0.000,B 0.000,C 90.000,E1 74.338} C_DIS
LIN {X 0.027,Y -476.755,Z 351.213,A 0.000,B 0.000,C 90.000,E1 74.338} C_DIS
LIN {X 0.029,Y -481.788,Z 351.208,A 0.000,B 0.000,C 90.000,E1 73.378} C_DIS
LIN {X -0.041,Y -487.046,Z 351.202,A 0.000,B 0.000,C 90.000,E1 72.308} C_DIS
LIN {X -0.031,Y -488.399,Z 351.200,A 0.000,B 0.000,C 90.000,E1 72.000} C_DIS
LIN {X -0.013,Y -489.964,Z 351.198,A 0.000,B 0.000,C 90.000,E1 71.692} C_DIS
LIN {X 0.100,Y -491.932,Z 351.196,A 0.000,B 0.000,C 90.000,E1 71.221} C_DIS
LIN {X 0.133,Y -493.242,Z 351.194,A 0.000,B 0.000,C 90.000,E1 70.913} C_DIS
LIN {X -0.107,Y -497.655,Z 351.188,A 0.000,B 0.000,C 90.000,E1 69.880} C_DIS
LIN {X 0.277,Y -500.570,Z 351.184,A 0.000,B 0.000,C 90.000,E1 69.082} C_DIS
LIN {X -0.080,Y -504.565,Z 351.177,A 0.000,B 0.000,C 90.000,E1 67.922} C_DIS
LIN {X -0.196,Y -508.305,Z 351.171,A 0.000,B 0.000,C 90.000,E1 66.741} C_DIS
LIN {X -0.049,Y -511.916,Z 351.164,A 0.000,B 0.000,C 90.000,E1 65.537} C_DIS
LIN {X 0.281,Y -516.209,Z 351.156,A 0.000,B 0.000,C 90.000,E1 64.024} C_DIS
LIN {X 0.088,Y -519.580,Z 351.149,A 0.000,B 0.000,C 90.000,E1 62.871} C_DIS
LIN {X 0.002,Y -524.472,Z 351.140,A 0.000,B 0.000,C 90.000,E1 61.129} C_DIS
LIN {X 0.228,Y -530.144,Z 351.128,A 0.000,B 0.000,C 90.000,E1 59.076} C_DIS
LIN {X -0.020,Y -535.729,Z 351.117,A 0.000,B 0.000,C 90.000,E1 57.089} C_DIS
LIN {X 0.133,Y -537.986,Z 351.112,A 0.000,B 0.000,C 90.000,E1 56.215} C_DIS
LIN {X -0.107,Y -541.662,Z 351.105,A 0.000,B 0.000,C 90.000,E1 54.815} C_DIS
LIN {X -0.317,Y -544.358,Z 351.098,A 0.000,B 0.000,C 90.000,E1 53.703} C_DIS
LIN {X -0.130,Y -547.436,Z 351.090,A 0.000,B 0.000,C 90.000,E1 52.271} C_DIS
LIN {X 0.023,Y -550.139,Z 351.083,A 0.000,B 0.000,C 90.000,E1 50.848} C_DIS
LIN {X 0.186,Y -551.467,Z 351.078,A 0.000,B 0.000,C 90.000,E1 49.989} C_DIS
LIN {X -0.123,Y -552.251,Z 351.075,A 0.000,B 0.000,C 90.000,E1 49.461} C_DIS
LIN {X -0.006,Y -553.186,Z 351.070,A 0.000,B 0.000,C 90.000,E1 48.609} C_DIS
LIN {X 0.126,Y -553.843,Z 351.065,A 0.000,B 0.000,C 90.000,E1 47.757} C_DIS
LIN {X -0.083,Y -554.422,Z 351.059,A 0.000,B 0.000,C 90.000,E1 46.662} C_DIS
LIN {X 0.147,Y -554.222,Z 351.051,A 0.000,B 0.000,C 90.000,E1 45.243} C_DIS
LIN {X 0.321,Y -553.732,Z 351.045,A 0.000,B 0.000,C 90.000,E1 44.109} C_DIS
LIN {X 0.053,Y -553.154,Z 351.041,A 0.000,B 0.000,C 90.000,E1 43.299} C_DIS
LIN {X -0.176,Y -552.071,Z 351.034,A 0.000,B 0.000,C 90.000,E1 42.204} C_DIS
LIN {X 0.044,Y -550.441,Z 351.027,A 0.000,B 0.000,C 90.000,E1 40.782} C_DIS
LIN {X 0.190,Y -548.989,Z 351.020,A 0.000,B 0.000,C 90.000,E1 39.644} C_DIS
LIN {X 0.012,Y -547.085,Z 351.013,A 0.000,B 0.000,C 90.000,E1 38.257} C_DIS
LIN {X -0.159,Y -544.884,Z 351.003,A 0.000,B 0.000,C 90.000,E1 36.583} C_DIS
LIN {X -0.210,Y -541.938,Z 350.991,A 0.000,B 0.000,C 90.000,E1 34.326} C_DIS
LIN {X 0.244,Y -539.170,Z 350.978,A 0.000,B 0.000,C 90.000,E1 32.005} C_DIS
LIN {X 0.056,Y -536.552,Z 350.965,A 0.000,B 0.000,C 90.000,E1 29.745} C_DIS
LIN {X -0.188,Y -534.481,Z 350.954,A 0.000,B 0.000,C 90.000,E1 27.769} C_DIS
LIN {X 0.015,Y -532.654,Z 350.945,A 0.000,B 0.000,C 90.000,E1 26.027} C_DIS
LIN {X -0.283,Y -530.964,Z 350.935,A 0.000,B 0.000,C 90.000,E1 24.335} C_DIS
LIN {X 0.066,Y -529.211,Z 350.924,A 0.000,B 0.000,C 90.000,E1 22.280} C_DIS
LIN {X -0.002,Y -528.076,Z 350.916,A 0.000,B 0.000,C 90.000,E1 20.844} C_DIS
LIN {X -0.126,Y -526.773,Z 350.905,A 0.000,B 0.000,C 90.000,E1 18.833} C_DIS
LIN {X -0.108,Y -525.687,Z 350.893,A 0.000,B 0.000,C 90.000,E1 16.804} C_DIS
LIN {X -0.105,Y -524.992,Z 350.882,A 0.000,B 0.000,C 90.000,E1 14.773} C_DIS
LIN {X 0.284,Y -524.545,Z 350.866,A 0.000,B 0.000,C 90.000,E1 11.827} C_DIS
LIN {X -0.204,Y -524.755,Z 350.853,A 0.000,B 0.000,C 90.000,E1 9.557} C_DIS
LIN {X -0.246,Y -525.465,Z 350.840,A 0.000,B 0.000,C 90.000,E1 7.239} C_DIS
LIN {X 0.174,Y -526.499,Z 350.829,A 0.000,B 0.000,C 90.000,E1 5.163} C_DIS
LIN {X -0.045,Y -528.658,Z 350.813,A 0.000,B 0.000,C 90.000,E1 2.293} C_DIS
LIN {X 0.144,Y -533.182,Z 350.791,A 0.000,B 0.000,C 90.000,E1 358.339} C_DIS
LIN {X 0.188,Y -537.047,Z 350.777,A 0.000,B 0.000,C 90.000,E1 355.755} C_DIS
LIN {X -0.189,Y -540.488,Z 350.766,A 0.000,B 0.000,C 90.000,E1 353.799} C_DIS
LIN {X 0.124,Y -548.539,Z 350.743,A 0.000,B 0.000,C 90.000,E1 349.803} C_DIS
LIN {X -0.222,Y -559.634,Z 350.720,A 0.000,B 0.000,C 90.000,E1 345.644} C_DIS
LIN {X -0.141,Y -564.572,Z 350.711,A 0.000,B 0.000,C 90.000,E1 343.976} C_DIS
LIN {X 0.049,Y -569.782,Z 350.702,A 0.000,B 0.000,C 90.000,E1 342.308} C_DIS
LIN {X -0.184,Y -572.401,Z 350.697,A 0.000,B 0.000,C 90.000,E1 341.511} C_DIS
LIN {X 0.176,Y -578.518,Z 350.687,A 0.000,B 0.000,C 90.000,E1 339.571} C_DIS
LIN {X 0.080,Y -582.811,Z 350.679,A 0.000,B 0.000,C 90.000,E1 338.230} C_DIS
LIN {X -0.273,Y -587.149,Z 350.672,A 0.000,B 0.000,C 90.000,E1 336.922} C_DIS
LIN {X -0.224,Y -593.355,Z 350.661,A 0.000,B 0.000,C 90.000,E1 335.049} C_DIS
LIN {X -0.050,Y -599.704,Z 350.651,A 0.000,B 0.000,C 90.000,E1 333.179} C_DIS
LIN {X 0.237,Y -606.981,Z 350.639,A 0.000,B 0.000,C 90.000,E1 331.051} C_DIS
LIN {X -0.012,Y -613.431,Z 350.629,A 0.000,B 0.000,C 90.000,E1 329.253} C_DIS
LIN {X 0.136,Y -618.127,Z 350.622,A 0.000,B 0.000,C 90.000,E1 327.946} C_DIS
LIN {X 0.267,Y -625.394,Z 350.611,A 0.000,B 0.000,C 90.000,E1 325.881} C_DIS
LIN {X -0.278,Y -630.584,Z 350.602,A 0.000,B 0.000,C 90.000,E1 324.402} C_DIS
LIN {X -0.213,Y -634.810,Z 350.595,A 0.000,B 0.000,C 90.000,E1 323.130} C_DIS
LIN {X 0.306,Y -638.886,Z 350.588,A 0.000,B 0.000,C 90.000,E1 321.823} C_DIS
LIN {X -0.272,Y -646.210,Z 350.576,A 0.000,B 0.000,C 90.000,E1 319.622} C_DIS
LIN {X -0.067,Y -649.426,Z 350.570,A 0.000,B 0.000,C 90.000,E1 318.609} C_DIS
LIN {X -0.058,Y -658.369,Z 350.555,A 0.000,B 0.000,C 90.000,E1 315.891} C_DIS
LIN {X -0.156,Y -661.578,Z 350.550,A 0.000,B 0.000,C 90.000,E1 314.919} C_DIS
LIN {X -0.234,Y -667.123,Z 350.540,A 0.000,B 0.000,C 90.000,E1 313.218} C_DIS
LIN {X -0.175,Y -671.786,Z 350.532,A 0.000,B 0.000,C 90.000,E1 311.757} C_DIS
LIN {X -0.060,Y -674.671,Z 350.527,A 0.000,B 0.000,C 90.000,E1 310.782} C_DIS
LIN {X -0.290,Y -678.848,Z 350.519,A 0.000,B 0.000,C 90.000,E1 309.358} C_DIS
LIN {X -0.086,Y -681.505,Z 350.513,A 0.000,B 0.000,C 90.000,E1 308.382} C_DIS
LIN {X -0.274,Y -683.926,Z 350.508,A 0.000,B 0.000,C 90.000,E1 307.443} C_DIS
LIN {X -0.053,Y -685.614,Z 350.504,A 0.000,B 0.000,C 90.000,E1 306.710} C_DIS
LIN {X -0.227,Y -687.115,Z 350.500,A 0.000,B 0.000,C 90.000,E1 306.011} C_DIS
LIN {X -0.382,Y -688.496,Z 350.496,A 0.000,B 0.000,C 90.000,E1 305.311} C_DIS
LIN {X 0.043,Y -689.679,Z 350.492,A 0.000,B 0.000,C 90.000,E1 304.565} C_DIS
LIN {X -0.084,Y -690.743,Z 350.488,A 0.000,B 0.000,C 90.000,E1 303.865} C_DIS
LIN {X -0.205,Y -691.505,Z 350.484,A 0.000,B 0.000,C 90.000,E1 303.166} C_DIS
LIN {X -0.099,Y -692.185,Z 350.479,A 0.000,B 0.000,C 90.000,E1 302.212} C_DIS
LIN {X 0.139,Y -692.385,Z 350.476,A 0.000,B 0.000,C 90.000,E1 301.720} C_DIS
LIN {X 0.012,Y -692.485,Z 350.474,A 0.000,B 0.000,C 90.000,E1 301.258} C_DIS
LIN {X 0.125,Y -692.279,Z 350.470,A 0.000,B 0.000,C 90.000,E1 300.541} C_DIS
LIN {X 0.005,Y -691.969,Z 350.467,A 0.000,B 0.000,C 90.000,E1 300.079} C_DIS
LIN {X -0.241,Y -690.941,Z 350.462,A 0.000,B 0.000,C 90.000,E1 299.155} C_DIS
LIN {X -0.133,Y -689.908,Z 350.458,A 0.000,B 0.000,C 90.000,E1 298.437} C_DIS
LIN {X -0.183,Y -687.682,Z 350.451,A 0.000,B 0.000,C 90.000,E1 297.257} C_DIS
LIN {X 0.028,Y -685.186,Z 350.445,A 0.000,B 0.000,C 90.000,E1 296.052} C_DIS
LIN {X 0.281,Y -683.055,Z 350.440,A 0.000,B 0.000,C 90.000,E1 295.079} C_DIS
LIN {X 0.329,Y -679.563,Z 350.432,A 0.000,B 0.000,C 90.000,E1 293.643} C_DIS
LIN {X -0.056,Y -677.132,Z 350.426,A 0.000,B 0.000,C 90.000,E1 292.717} C_DIS
LIN {X -0.290,Y -673.945,Z 350.420,A 0.000,B 0.000,C 90.000,E1 291.535} C_DIS
LIN {X -0.035,Y -670.221,Z 350.411,A 0.000,B 0.000,C 90.000,E1 290.066} C_DIS
LIN {X -0.035,Y -665.297,Z 350.401,A 0.000,B 0.000,C 90.000,E1 288.127} C_DIS
LIN {X -0.366,Y -660.665,Z 350.390,A 0.000,B 0.000,C 90.000,E1 286.205} C_DIS
LIN {X 0.165,Y -655.969,Z 350.378,A 0.000,B 0.000,C 90.000,E1 283.953} C_DIS
LIN {X -0.008,Y -649.214,Z 350.356,A 0.000,B 0.000,C 90.000,E1 280.018} C_DIS
LIN {X -0.281,Y -645.186,Z 350.335,A 0.000,B 0.000,C 90.000,E1 276.315} C_DIS
LIN {X -0.261,Y -643.728,Z 350.323,A 0.000,B 0.000,C 90.000,E1 274.069} C_DIS
LIN {X 0.207,Y -642.808,Z 350.306,A 0.000,B 0.000,C 90.000,E1 271.031} C_DIS
LIN {X 0.220,Y -642.908,Z 350.291,A 0.000,B 0.000,C 90.000,E1 268.282} C_DIS
LIN {X -0.309,Y -643.644,Z 350.280,A 0.000,B 0.000,C 90.000,E1 266.331} C_DIS
LIN {X 0.116,Y -644.493,Z 350.270,A 0.000,B 0.000,C 90.000,E1 264.546} C_DIS
LIN {X -0.321,Y -645.570,Z 350.259,A 0.000,B 0.000,C 90.000,E1 262.591} C_DIS
LIN {X 0.313,Y -646.705,Z 350.249,A 0.000,B 0.000,C 90.000,E1 260.792} C_DIS
LIN {X 0.107,Y -647.422,Z 350.242,A 0.000,B 0.000,C 90.000,E1 259.567} C_DIS
LIN {X -0.269,Y -649.234,Z 350.228,A 0.000,B 0.000,C 90.000,E1 257.117} C_DIS
LIN {X -0.171,Y -649.890,Z 350.223,A 0.000,B 0.000,C 90.000,E1 256.117} C_DIS
LIN {X 0.063,Y -650.155,Z 350.219,A 0.000,B 0.000,C 90.000,E1 255.353} C_DIS
LIN {X -0.161,Y -650.182,Z 350.215,A 0.000,B 0.000,C 90.000,E1 254.629} C_DIS
LIN {X 0.070,Y -649.943,Z 350.210,A 0.000,B 0.000,C 90.000,E1 253.866} C_DIS
LIN {X -0.146,Y -649.516,Z 350.206,A 0.000,B 0.000,C 90.000,E1 253.142} C_DIS
LIN {X -0.281,Y -649.363,Z 350.205,A 0.000,B 0.000,C 90.000,E1 252.906} C_DIS
LIN {X -0.224,Y -649.009,Z 350.204,A 0.000,B 0.000,C 90.000,E1 252.653} C_DIS
LIN {X 0.178,Y -648.344,Z 350.199,A 0.000,B 0.000,C 90.000,E1 251.873} C_DIS
LIN {X -0.044,Y -647.290,Z 350.195,A 0.000,B 0.000,C 90.000,E1 251.148} C_DIS
LIN {X -0.277,Y -645.953,Z 350.191,A 0.000,B 0.000,C 90.000,E1 250.423} C_DIS
LIN {X 0.238,Y -644.931,Z 350.188,A 0.000,B 0.000,C 90.000,E1 249.880} C_DIS
LIN {X -0.028,Y -643.098,Z 350.184,A 0.000,B 0.000,C 90.000,E1 249.156} C_DIS
LIN {X -0.025,Y -640.182,Z 350.179,A 0.000,B 0.000,C 90.000,E1 248.156} C_DIS
LIN {X -0.154,Y -638.588,Z 350.176,A 0.000,B 0.000,C 90.000,E1 247.667} C_DIS
LIN {X -0.201,Y -635.041,Z 350.170,A 0.000,B 0.000,C 90.000,E1 246.666} C_DIS
LIN {X -0.292,Y -631.437,Z 350.165,A 0.000,B 0.000,C 90.000,E1 245.665} C_DIS
LIN {X 0.132,Y -627.675,Z 350.159,A 0.000,B 0.000,C 90.000,E1 244.613} C_DIS
LIN {X 0.199,Y -623.729,Z 350.153,A 0.000,B 0.000,C 90.000,E1 243.589} C_DIS
LIN {X -0.348,Y -617.771,Z 350.145,A 0.000,B 0.000,C 90.000,E1 242.103} C_DIS
LIN {X -0.145,Y -612.791,Z 350.138,A 0.000,B 0.000,C 90.000,E1 240.795} C_DIS
LIN {X 0.168,Y -605.725,Z 350.128,A 0.000,B 0.000,C 90.000,E1 238.948} C_DIS
LIN {X 0.104,Y -598.799,Z 350.117,A 0.000,B 0.000,C 90.000,E1 237.120} C_DIS
LIN {X -0.404,Y -587.523,Z 350.100,A 0.000,B 0.000,C 90.000,E1 233.989} C_DIS
LIN {X 0.185,Y -584.863,Z 350.095,A 0.000,B 0.000,C 90.000,E1 233.130} C_DIS
LIN {X -0.183,Y -579.940,Z 350.088,A 0.000,B 0.000,C 90.000,E1 231.823} C_DIS
LIN {X -0.301,Y -569.487,Z 350.071,A 0.000,B 0.000,C 90.000,E1 228.852} C_DIS
LIN {X -0.194,Y -565.020,Z 350.064,A 0.000,B 0.000,C 90.000,E1 227.472} C_DIS
LIN {X 0.210,Y -560.483,Z 350.056,A 0.000,B 0.000,C 90.000,E1 226.053} C_DIS
LIN {X 0.131,Y -555.932,Z 350.048,A 0.000,B 0.000,C 90.000,E1 224.676} C_DIS
LIN {X -0.030,Y -551.454,Z 350.041,A 0.000,B 0.000,C 90.000,E1 223.299} C_DIS
LIN {X -0.245,Y -546.979,Z 350.033,A 0.000,B 0.000,C 90.000,E1 221.919} C_DIS
LIN {X 0.259,Y -541.692,Z 350.023,A 0.000,B 0.000,C 90.000,E1 220.172} C_DIS
LIN {X -0.114,Y -534.793,Z 350.011,A 0.000,B 0.000,C 90.000,E1 217.935} C_DIS
LIN {X 0.252,Y -528.162,Z 349.998,A 0.000,B 0.000,C 90.000,E1 215.598} C_DIS
LIN {X 0.171,Y -522.662,Z 349.987,A 0.000,B 0.000,C 90.000,E1 213.579} C_DIS
LIN {X 0.055,Y -515.531,Z 349.970,A 0.000,B 0.000,C 90.000,E1 210.669} C_DIS
LIN {X 0.075,Y -510.262,Z 349.957,A 0.000,B 0.000,C 90.000,E1 208.309} C_DIS
LIN {X 0.064,Y -505.709,Z 349.946,A 0.000,B 0.000,C 90.000,E1 206.232} C_DIS
LIN {X -0.212,Y -502.500,Z 349.938,A 0.000,B 0.000,C 90.000,E1 204.771} C_DIS
LIN {X -0.164,Y -499.827,Z 349.931,A 0.000,B 0.000,C 90.000,E1 203.567} C_DIS
LIN {X 0.162,Y -496.457,Z 349.923,A 0.000,B 0.000,C 90.000,E1 202.025} C_DIS
LIN {X -0.211,Y -493.002,Z 349.914,A 0.000,B 0.000,C 90.000,E1 200.556} C_DIS
LIN {X -0.127,Y -488.151,Z 349.902,A 0.000,B 0.000,C 90.000,E1 198.417} C_DIS
LIN {X -0.026,Y -482.971,Z 349.889,A 0.000,B 0.000,C 90.000,E1 195.953} C_DIS
LIN {X 0.000,Y -478.090,Z 349.875,A 0.000,B 0.000,C 90.000,E1 193.480} C_DIS
LIN {X -0.192,Y -475.182,Z 349.866,A 0.000,B 0.000,C 90.000,E1 191.951} C_DIS
LIN {X 0.138,Y -471.139,Z 349.854,A 0.000,B 0.000,C 90.000,E1 189.726} C_DIS
LIN {X 0.120,Y -467.400,Z 349.842,A 0.000,B 0.000,C 90.000,E1 187.530} C_DIS
LIN {X 0.007,Y -463.928,Z 349.830,A 0.000,B 0.000,C 90.000,E1 185.334} C_DIS
LIN {X -0.199,Y -458.948,Z 349.809,A 0.000,B 0.000,C 90.000,E1 181.547} C_DIS
LIN {X -0.016,Y -455.163,Z 349.785,A 0.000,B 0.000,C 90.000,E1 177.364} C_DIS
LIN {X 0.008,Y -453.537,Z 349.768,A 0.000,B 0.000,C 90.000,E1 174.147} C_DIS
LIN {X -0.131,Y -453.050,Z 349.748,A 0.000,B 0.000,C 90.000,E1 170.622} C_DIS
LIN {X 0.050,Y -453.513,Z 349.732,A 0.000,B 0.000,C 90.000,E1 167.701} C_DIS
LIN {X 0.084,Y -456.042,Z 349.707,A 0.000,B 0.000,C 90.000,E1 163.196} C_DIS
LIN {X -0.007,Y -461.066,Z 349.680,A 0.000,B 0.000,C 90.000,E1 158.411} C_DIS
LIN {X -0.009,Y -466.331,Z 349.661,A 0.000,B 0.000,C 90.000,E1 154.921} C_DIS
LIN {X 0.025,Y -472.372,Z 349.643,A 0.000,B 0.000,C 90.000,E1 151.769} C_DIS
LIN {X -0.115,Y -482.207,Z 349.621,A 0.000,B 0.000,C 90.000,E1 147.740} C_DIS
LIN {X -0.282,Y -491.326,Z 349.604,A 0.000,B 0.000,C 90.000,E1 144.689} C_DIS
LIN {X 0.055,Y -496.196,Z 349.595,A 0.000,B 0.000,C 90.000,E1 143.130} C_DIS
LIN {X -0.051,Y -499.245,Z 349.590,A 0.000,B 0.000,C 90.000,E1 142.236} C_DIS
LIN {X 0.157,Y -503.153,Z 349.584,A 0.000,B 0.000,C 90.000,E1 141.009} C_DIS
LIN {X 0.027,Y -506.849,Z 349.577,A 0.000,B 0.000,C 90.000,E1 139.828} C_DIS
LIN {X 0.182,Y -511.219,Z 349.569,A 0.000,B 0.000,C 90.000,E1 138.324} C_DIS
LIN {X -0.139,Y -513.634,Z 349.564,A 0.000,B 0.000,C 90.000,E1 137.472} C_DIS
LIN {X -0.083,Y -515.730,Z 349.559,A 0.000,B 0.000,C 90.000,E1 136.581} C_DIS
LIN {X 0.013,Y -517.568,Z 349.554,A 0.000,B 0.000,C 90.000,E1 135.688} C_DIS
LIN {X -0.253,Y -519.059,Z 349.549,A 0.000,B 0.000,C 90.000,E1 134.838} C_DIS
LIN {X -0.133,Y -520.165,Z 349.544,A 0.000,B 0.000,C 90.000,E1 133.947} C_DIS
LIN {X -0.005,Y -520.973,Z 349.539,A 0.000,B 0.000,C 90.000,E1 133.056} C_DIS
LIN {X 0.221,Y -521.187,Z 349.536,A 0.000,B 0.000,C 90.000,E1 132.447} C_DIS
LIN {X 0.160,Y -521.438,Z 349.534,A 0.000,B 0.000,C 90.000,E1 132.162} C_DIS
LIN {X 0.238,Y -521.647,Z 349.528,A 0.000,B 0.000,C 90.000,E1 130.987} C_DIS
LIN {X -0.316,Y -521.383,Z 349.523,A 0.000,B 0.000,C 90.000,E1 130.172} C_DIS
LIN {X -0.083,Y -521.052,Z 349.520,A 0.000,B 0.000,C 90.000,E1 129.564} C_DIS
LIN {X 0.038,Y -519.878,Z 349.513,A 0.000,B 0.000,C 90.000,E1 128.382} C_DIS
LIN {X -0.122,Y -518.787,Z 349.508,A 0.000,B 0.000,C 90.000,E1 127.523} C_DIS
LIN {X 0.311,Y -516.826,Z 349.500,A 0.000,B 0.000,C 90.000,E1 126.011} C_DIS
LIN {X -0.250,Y -515.015,Z 349.494,A 0.000,B 0.000,C 90.000,E1 124.898} C_DIS
LIN {X -0.118,Y -513.015,Z 349.487,A 0.000,B 0.000,C 90.000,E1 123.706} C_DIS
LIN {X 0.127,Y -510.760,Z 349.481,A 0.000,B 0.000,C 90.000,E1 122.498} C_DIS
LIN {X -0.090,Y -508.231,Z 349.474,A 0.000,B 0.000,C 90.000,E1 121.337} C_DIS
LIN {X -0.288,Y -504.876,Z 349.466,A 0.000,B 0.000,C 90.000,E1 119.873} C_DIS
LIN {X 0.267,Y -501.998,Z 349.459,A 0.000,B 0.000,C 90.000,E1 118.615} C_DIS
LIN {X -0.247,Y -497.411,Z 349.449,A 0.000,B 0.000,C 90.000,E1 116.873} C_DIS
LIN {X -0.055,Y -494.159,Z 349.442,A 0.000,B 0.000,C 90.000,E1 115.643} C_DIS
LIN {X 0.030,Y -492.544,Z 349.439,A 0.000,B 0.000,C 90.000,E1 115.027} C_DIS
LIN {X -0.101,Y -489.889,Z 349.434,A 0.000,B 0.000,C 90.000,E1 114.131} C_DIS
LIN {X 0.008,Y -486.152,Z 349.427,A 0.000,B 0.000,C 90.000,E1 112.898} C_DIS
LIN {X 0.074,Y -481.312,Z 349.419,A 0.000,B 0.000,C 90.000,E1 111.354} C_DIS
LIN {X 0.057,Y -476.995,Z 349.412,A 0.000,B 0.000,C 90.000,E1 110.120} C_DIS
LIN {X -0.161,Y -473.537,Z 349.407,A 0.000,B 0.000,C 90.000,E1 109.214} C_DIS
LIN {X -0.062,Y -467.413,Z 349.398,A 0.000,B 0.000,C 90.000,E1 107.638} C_DIS
LIN {X 0.014,Y -463.516,Z 349.393,A 0.000,B 0.000,C 90.000,E1 106.677} C_DIS
LIN {X -0.027,Y -463.527,Z 349.393,A 0.000,B 0.000,C 90.000,E1 106.677} C_DIS
LIN {X -0.270,Y -467.268,Z 349.384,A 0.000,B 0.000,C 90.000,E1 105.134} C_DIS
LIN {X 0.106,Y -467.962,Z 349.382,A 0.000,B 0.000,C 90.000,E1 104.773} C_DIS
LIN {X 0.070,Y -476.180,Z 349.356,A 0.000,B 0.000,C 90.000,E1 100.074} C_DIS
LIN {X -0.154,Y -482.086,Z 349.330,A 0.000,B 0.000,C 90.000,E1 95.448} C_DIS
LIN {X 0.076,Y -485.505,Z 349.305,A 0.000,B 0.000,C 90.000,E1 90.802} C_DIS
LIN {X 0.108,Y -486.383,Z 349.281,A 0.000,B 0.000,C 90.000,E1 86.502} C_DIS
LIN {X -0.067,Y -486.361,Z 349.279,A 0.000,B 0.000,C 90.000,E1 86.216} C_DIS
LIN {X 0.016,Y -484.684,Z 349.253,A 0.000,B 0.000,C 90.000,E1 81.602} C_DIS
LIN {X -0.084,Y -480.607,Z 349.228,A 0.000,B 0.000,C 90.000,E1 76.992} C_DIS
LIN {X 0.241,Y -480.245,Z 349.226,A 0.000,B 0.000,C 90.000,E1 76.645} C_DIS
LIN {X 0.031,Y -476.891,Z 349.214,A 0.000,B 0.000,C 90.000,E1 74.448} C_DIS
LIN {X -0.010,Y -476.898,Z 349.214,A 0.000,B 0.000,C 90.000,E1 74.448} C_DIS
LIN {X -0.107,Y -482.090,Z 349.208,A 0.000,B 0.000,C 90.000,E1 73.433} C_DIS
LIN {X -0.033,Y -485.751,Z 349.204,A 0.000,B 0.000,C 90.000,E1 72.653} C_DIS
LIN {X 0.065,Y -487.833,Z 349.201,A 0.000,B 0.000,C 90.000,E1 72.181} C_DIS
LIN {X -0.054,Y -490.507,Z 349.198,A 0.000,B 0.000,C 90.000,E1 71.583} C_DIS
LIN {X -0.028,Y -491.690,Z 349.196,A 0.000,B 0.000,C 90.000,E1 71.275} C_DIS
LIN {X 0.088,Y -493.383,Z 349.194,A 0.000,B 0.000,C 90.000,E1 70.859} C_DIS
LIN {X 0.099,Y -498.126,Z 349.187,A 0.000,B 0.000,C 90.000,E1 69.645} C_DIS
LIN {X -0.248,Y -500.325,Z 349.184,A 0.000,B 0.000,C 90.000,E1 69.082} C_DIS
LIN {X 0.127,Y -505.139,Z 349.175,A 0.000,B 0.000,C 90.000,E1 67.539} C_DIS
LIN {X 0.025,Y -508.809,Z 349.169,A 0.000,B 0.000,C 90.000,E1 66.357} C_DIS
LIN {X -0.030,Y -512.304,Z 349.162,A 0.000,B 0.000,C 90.000,E1 65.177} C_DIS
LIN {X -0.285,Y -515.728,Z 349.156,A 0.000,B 0.000,C 90.000,E1 64.024} C_DIS
LIN {X -0.027,Y -519.102,Z 349.149,A 0.000,B 0.000,C 90.000,E1 62.820} C_DIS
LIN {X 0.121,Y -523.993,Z 349.139,A 0.000,B 0.000,C 90.000,E1 61.051} C_DIS
LIN {X 0.343,Y -529.703,Z 349.128,A 0.000,B 0.000,C 90.000,E1 58.997} C_DIS
LIN {X -0.189,Y -534.523,Z 349.118,A 0.000,B 0.000,C 90.000,E1 57.327} C_DIS
LIN {X -0.056,Y -537.608,Z 349.112,A 0.000,B 0.000,C 90.000,E1 56.167} C_DIS
LIN {X -0.017,Y -540.556,Z 349.106,A 0.000,B 0.000,C 90.000,E1 55.022} C_DIS
LIN {X -0.241,Y -543.344,Z 349.099,A 0.000,B 0.000,C 90.000,E1 53.909} C_DIS
LIN {X -0.070,Y -546.521,Z 349.092,A 0.000,B 0.000,C 90.000,E1 52.477} C_DIS
LIN {X -0.276,Y -549.328,Z 349.084,A 0.000,B 0.000,C 90.000,E1 51.090} C_DIS
LIN {X 0.282,Y -551.234,Z 349.077,A 0.000,B 0.000,C 90.000,E1 49.908} C_DIS
LIN {X -0.333,Y -552.745,Z 349.071,A 0.000,B 0.000,C 90.000,E1 48.852} C_DIS
LIN {X -0.209,Y -553.582,Z 349.067,A 0.000,B 0.000,C 90.000,E1 48.000} C_DIS
LIN {X 0.011,Y -554.478,Z 349.059,A 0.000,B 0.000,C 90.000,E1 46.581} C_DIS
LIN {X 0.064,Y -554.616,Z 349.057,A 0.000,B 0.000,C 90.000,E1 46.296} C_DIS
LIN {X 0.244,Y -554.595,Z 349.051,A 0.000,B 0.000,C 90.000,E1 45.162} C_DIS
LIN {X -0.359,Y -554.210,Z 349.045,A 0.000,B 0.000,C 90.000,E1 44.109} C_DIS
LIN {X 0.160,Y -553.667,Z 349.040,A 0.000,B 0.000,C 90.000,E1 43.218} C_DIS
LIN {X -0.081,Y -552.929,Z 349.036,A 0.000,B 0.000,C 90.000,E1 42.405} C_DIS
LIN {X 0.111,Y -551.385,Z 349.028,A 0.000,B 0.000,C 90.000,E1 40.987} C_DIS
LIN {X -0.086,Y -549.982,Z 349.022,A 0.000,B 0.000,C 90.000,E1 39.886} C_DIS
LIN {X 0.100,Y -548.146,Z 349.014,A 0.000,B 0.000,C 90.000,E1 38.463} C_DIS
LIN {X -0.010,Y -545.563,Z 349.003,A 0.000,B 0.000,C 90.000,E1 36.503} C_DIS
LIN {X -0.076,Y -543.002,Z 348.992,A 0.000,B 0.000,C 90.000,E1 34.532} C_DIS
LIN {X -0.062,Y -540.566,Z 348.981,A 0.000,B 0.000,C 90.000,E1 32.546} C_DIS
LIN {X 0.067,Y -538.256,Z 348.970,A 0.000,B 0.000,C 90.000,E1 30.541} C_DIS
LIN {X -0.044,Y -536.717,Z 348.962,A 0.000,B 0.000,C 90.000,E1 29.127} C_DIS
LIN {X -0.236,Y -535.271,Z 348.954,A 0.000,B 0.000,C 90.000,E1 27.719} C_DIS
LIN {X -0.008,Y -533.457,Z 348.944,A 0.000,B 0.000,C 90.000,E1 25.976} C_DIS
LIN {X -0.063,Y -531.807,Z 348.935,A 0.000,B 0.000,C 90.000,E1 24.259} C_DIS
LIN {X 0.298,Y -530.062,Z 348.924,A 0.000,B 0.000,C 90.000,E1 22.206} C_DIS
LIN {X 0.232,Y -528.728,Z 348.914,A 0.000,B 0.000,C 90.000,E1 20.482} C_DIS
LIN {X -0.041,Y -527.498,Z 348.903,A 0.000,B 0.000,C 90.000,E1 18.489} C_DIS
LIN {X 0.178,Y -526.418,Z 348.890,A 0.000,B 0.000,C 90.000,E1 16.150} C_DIS
LIN {X 0.213,Y -525.713,Z 348.877,A 0.000,B 0.000,C 90.000,E1 13.828} C_DIS
LIN {X -0.033,Y -525.484,Z 348.864,A 0.000,B 0.000,C 90.000,E1 11.535} C_DIS
LIN {X 0.024,Y -525.805,Z 348.851,A 0.000,B 0.000,C 90.000,E1 9.208} C_DIS
LIN {X -0.024,Y -526.894,Z 348.835,A 0.000,B 0.000,C 90.000,E1 6.315} C_DIS
LIN {X -0.143,Y -528.013,Z 348.824,A 0.000,B 0.000,C 90.000,E1 4.302} C_DIS
LIN {X 0.224,Y -530.459,Z 348.808,A 0.000,B 0.000,C 90.000,E1 1.375} C_DIS
LIN {X 0.161,Y -534.090,Z 348.791,A 0.000,B 0.000,C 90.000,E1 358.339} C_DIS
LIN {X 0.195,Y -537.469,Z 348.778,A 0.000,B 0.000,C 90.000,E1 356.045} C_DIS
LIN {X -0.244,Y -539.819,Z 348.770,A 0.000,B 0.000,C 90.000,E1 354.666} C_DIS
LIN {X 0.127,Y -548.612,Z 348.745,A 0.000,B 0.000,C 90.000,E1 350.095} C_DIS
LIN {X -0.169,Y -554.021,Z 348.733,A 0.000,B 0.000,C 90.000,E1 347.881} C_DIS
LIN {X -0.078,Y -560.317,Z 348.720,A 0.000,B 0.000,C 90.000,E1 345.644} C_DIS
LIN {X -0.051,Y -566.939,Z 348.708,A 0.000,B 0.000,C 90.000,E1 343.433} C_DIS
LIN {X 0.191,Y -572.222,Z 348.699,A 0.000,B 0.000,C 90.000,E1 341.764} C_DIS
LIN {X -0.166,Y -579.157,Z 348.687,A 0.000,B 0.000,C 90.000,E1 339.625} C_DIS
LIN {X -0.249,Y -583.454,Z 348.679,A 0.000,B 0.000,C 90.000,E1 338.284} C_DIS
LIN {X -0.047,Y -587.803,Z 348.672,A 0.000,B 0.000,C 90.000,E1 336.922} C_DIS
LIN {X -0.077,Y -594.908,Z 348.660,A 0.000,B 0.000,C 90.000,E1 334.793} C_DIS
LIN {X 0.139,Y -601.264,Z 348.650,A 0.000,B 0.000,C 90.000,E1 332.922} C_DIS
LIN {X -0.009,Y -607.663,Z 348.639,A 0.000,B 0.000,C 90.000,E1 331.101} C_DIS
LIN {X -0.021,Y -614.170,Z 348.629,A 0.000,B 0.000,C 90.000,E1 329.282} C_DIS
LIN {X -0.069,Y -618.850,Z 348.622,A 0.000,B 0.000,C 90.000,E1 327.995} C_DIS
LIN {X -0.034,Y -623.343,Z 348.615,A 0.000,B 0.000,C 90.000,E1 326.707} C_DIS
LIN {X 0.080,Y -626.896,Z 348.609,A 0.000,B 0.000,C 90.000,E1 325.674} C_DIS
LIN {X 0.081,Y -631.166,Z 348.602,A 0.000,B 0.000,C 90.000,E1 324.402} C_DIS
LIN {X 0.029,Y -636.088,Z 348.594,A 0.000,B 0.000,C 90.000,E1 322.889} C_DIS
LIN {X 0.184,Y -640.108,Z 348.587,A 0.000,B 0.000,C 90.000,E1 321.618} C_DIS
LIN {X 0.126,Y -646.629,Z 348.576,A 0.000,B 0.000,C 90.000,E1 319.622} C_DIS
LIN {X 0.402,Y -649.054,Z 348.572,A 0.000,B 0.000,C 90.000,E1 318.852} C_DIS
LIN {X -0.009,Y -656.197,Z 348.559,A 0.000,B 0.000,C 90.000,E1 316.662} C_DIS
LIN {X 0.341,Y -659.589,Z 348.554,A 0.000,B 0.000,C 90.000,E1 315.648} C_DIS
LIN {X 0.235,Y -664.246,Z 348.546,A 0.000,B 0.000,C 90.000,E1 314.190} C_DIS
LIN {X -0.247,Y -668.182,Z 348.539,A 0.000,B 0.000,C 90.000,E1 313.014} C_DIS
LIN {X 0.289,Y -672.785,Z 348.531,A 0.000,B 0.000,C 90.000,E1 311.515} C_DIS
LIN {X -0.003,Y -676.218,Z 348.524,A 0.000,B 0.000,C 90.000,E1 310.334} C_DIS
LIN {X -0.205,Y -680.262,Z 348.516,A 0.000,B 0.000,C 90.000,E1 308.910} C_DIS
LIN {X 0.014,Y -682.693,Z 348.511,A 0.000,B 0.000,C 90.000,E1 307.935} C_DIS
LIN {X -0.161,Y -685.022,Z 348.505,A 0.000,B 0.000,C 90.000,E1 306.996} C_DIS
LIN {X 0.243,Y -686.956,Z 348.500,A 0.000,B 0.000,C 90.000,E1 306.011} C_DIS
LIN {X 0.086,Y -688.287,Z 348.496,A 0.000,B 0.000,C 90.000,E1 305.311} C_DIS
LIN {X -0.057,Y -689.408,Z 348.492,A 0.000,B 0.000,C 90.000,E1 304.612} C_DIS
LIN {X -0.191,Y -690.406,Z 348.488,A 0.000,B 0.000,C 90.000,E1 303.913} C_DIS
LIN {X 0.258,Y -691.103,Z 348.484,A 0.000,B 0.000,C 90.000,E1 303.166} C_DIS
LIN {X 0.359,Y -691.676,Z 348.479,A 0.000,B 0.000,C 90.000,E1 302.212} C_DIS
LIN {X 0.000,Y -691.815,Z 348.478,A 0.000,B 0.000,C 90.000,E1 302.005} C_DIS
LIN {X 0.104,Y -691.873,Z 348.474,A 0.000,B 0.000,C 90.000,E1 301.288} C_DIS
LIN {X -0.025,Y -691.577,Z 348.470,A 0.000,B 0.000,C 90.000,E1 300.590} C_DIS
LIN {X -0.153,Y -691.257,Z 348.467,A 0.000,B 0.000,C 90.000,E1 300.129} C_DIS
LIN {X 0.189,Y -690.172,Z 348.462,A 0.000,B 0.000,C 90.000,E1 299.155} C_DIS
LIN {X -0.317,Y -689.135,Z 348.458,A 0.000,B 0.000,C 90.000,E1 298.487} C_DIS
LIN {X 0.225,Y -686.878,Z 348.452,A 0.000,B 0.000,C 90.000,E1 297.257} C_DIS
LIN {X -0.194,Y -684.342,Z 348.445,A 0.000,B 0.000,C 90.000,E1 296.104} C_DIS
LIN {X -0.246,Y -682.179,Z 348.440,A 0.000,B 0.000,C 90.000,E1 295.155} C_DIS
LIN {X 0.070,Y -678.650,Z 348.432,A 0.000,B 0.000,C 90.000,E1 293.695} C_DIS
LIN {X -0.148,Y -675.551,Z 348.425,A 0.000,B 0.000,C 90.000,E1 292.514} C_DIS
LIN {X 0.359,Y -669.821,Z 348.413,A 0.000,B 0.000,C 90.000,E1 290.301} C_DIS
LIN {X 0.247,Y -664.266,Z 348.401,A 0.000,B 0.000,C 90.000,E1 288.127} C_DIS
LIN {X -0.012,Y -660.160,Z 348.391,A 0.000,B 0.000,C 90.000,E1 286.441} C_DIS
LIN {X 0.080,Y -656.422,Z 348.382,A 0.000,B 0.000,C 90.000,E1 284.717} C_DIS
LIN {X -0.074,Y -652.958,Z 348.372,A 0.000,B 0.000,C 90.000,E1 283.008} C_DIS
LIN {X -0.098,Y -647.795,Z 348.354,A 0.000,B 0.000,C 90.000,E1 279.792} C_DIS
LIN {X 0.242,Y -644.527,Z 348.338,A 0.000,B 0.000,C 90.000,E1 276.777} C_DIS
LIN {X 0.010,Y -642.816,Z 348.324,A 0.000,B 0.000,C 90.000,E1 274.302} C_DIS
LIN {X 0.242,Y -641.760,Z 348.306,A 0.000,B 0.000,C 90.000,E1 271.031} C_DIS
LIN {X -0.235,Y -642.032,Z 348.288,A 0.000,B 0.000,C 90.000,E1 267.822} C_DIS
LIN {X 0.062,Y -642.683,Z 348.278,A 0.000,B 0.000,C 90.000,E1 266.045} C_DIS
LIN {X 0.061,Y -643.454,Z 348.270,A 0.000,B 0.000,C 90.000,E1 264.546} C_DIS
LIN {X 0.071,Y -644.699,Z 348.257,A 0.000,B 0.000,C 90.000,E1 262.299} C_DIS
LIN {X 0.053,Y -645.881,Z 348.248,A 0.000,B 0.000,C 90.000,E1 260.557} C_DIS
LIN {X -0.221,Y -647.420,Z 348.235,A 0.000,B 0.000,C 90.000,E1 258.342} C_DIS
LIN {X 0.074,Y -648.696,Z 348.227,A 0.000,B 0.000,C 90.000,E1 256.825} C_DIS
LIN {X -0.198,Y -649.108,Z 348.224,A 0.000,B 0.000,C 90.000,E1 256.353} C_DIS
LIN {X 0.029,Y -649.483,Z 348.220,A 0.000,B 0.000,C 90.000,E1 255.589} C_DIS
LIN {X -0.072,Y -649.678,Z 348.217,A 0.000,B 0.000,C 90.000,E1 255.102} C_DIS
LIN {X 0.292,Y -649.788,Z 348.215,A 0.000,B 0.000,C 90.000,E1 254.574} C_DIS
LIN {X 0.026,Y -649.771,Z 348.212,A 0.000,B 0.000,C 90.000,E1 254.102} C_DIS
LIN {X -0.326,Y -649.415,Z 348.206,A 0.000,B 0.000,C 90.000,E1 253.142} C_DIS
LIN {X 0.077,Y -648.917,Z 348.202,A 0.000,B 0.000,C 90.000,E1 252.362} C_DIS
LIN {X -0.143,Y -648.161,Z 348.198,A 0.000,B 0.000,C 90.000,E1 251.638} C_DIS
LIN {X -0.223,Y -647.587,Z 348.195,A 0.000,B 0.000,C 90.000,E1 251.148} C_DIS
LIN {X 0.155,Y -646.339,Z 348.191,A 0.000,B 0.000,C 90.000,E1 250.369} C_DIS
LIN {X -0.095,Y -644.765,Z 348.187,A 0.000,B 0.000,C 90.000,E1 249.645} C_DIS
LIN {X -0.134,Y -642.908,Z 348.183,A 0.000,B 0.000,C 90.000,E1 248.901} C_DIS
LIN {X -0.128,Y -640.057,Z 348.177,A 0.000,B 0.000,C 90.000,E1 247.901} C_DIS
LIN {X -0.257,Y -638.444,Z 348.174,A 0.000,B 0.000,C 90.000,E1 247.411} C_DIS
LIN {X 0.109,Y -633.308,Z 348.166,A 0.000,B 0.000,C 90.000,E1 245.869} C_DIS
LIN {X 0.252,Y -629.734,Z 348.160,A 0.000,B 0.000,C 90.000,E1 244.845} C_DIS
LIN {X 0.077,Y -625.871,Z 348.155,A 0.000,B 0.000,C 90.000,E1 243.845} C_DIS
LIN {X 0.123,Y -620.956,Z 348.148,A 0.000,B 0.000,C 90.000,E1 242.564} C_DIS
LIN {X -0.167,Y -616.074,Z 348.141,A 0.000,B 0.000,C 90.000,E1 241.307} C_DIS
LIN {X 0.042,Y -612.120,Z 348.135,A 0.000,B 0.000,C 90.000,E1 240.255} C_DIS
LIN {X -0.175,Y -605.140,Z 348.125,A 0.000,B 0.000,C 90.000,E1 238.456} C_DIS
LIN {X 0.351,Y -599.213,Z 348.116,A 0.000,B 0.000,C 90.000,E1 236.834} C_DIS
LIN {X -0.341,Y -588.911,Z 348.100,A 0.000,B 0.000,C 90.000,E1 233.989} C_DIS
LIN {X 0.263,Y -586.210,Z 348.095,A 0.000,B 0.000,C 90.000,E1 233.130} C_DIS
LIN {X 0.015,Y -583.262,Z 348.091,A 0.000,B 0.000,C 90.000,E1 232.351} C_DIS
LIN {X 0.011,Y -575.386,Z 348.079,A 0.000,B 0.000,C 90.000,E1 230.194} C_DIS
LIN {X 0.171,Y -568.184,Z 348.067,A 0.000,B 0.000,C 90.000,E1 228.000} C_DIS
LIN {X -0.071,Y -562.731,Z 348.058,A 0.000,B 0.000,C 90.000,E1 226.377} C_DIS
LIN {X -0.109,Y -558.175,Z 348.050,A 0.000,B 0.000,C 90.000,E1 225.000} C_DIS
LIN {X -0.227,Y -553.691,Z 348.042,A 0.000,B 0.000,C 90.000,E1 223.623} C_DIS
LIN {X 0.014,Y -548.332,Z 348.033,A 0.000,B 0.000,C 90.000,E1 221.919} C_DIS
LIN {X -0.221,Y -543.006,Z 348.024,A 0.000,B 0.000,C 90.000,E1 220.253} C_DIS
LIN {X -0.137,Y -536.965,Z 348.013,A 0.000,B 0.000,C 90.000,E1 218.257} C_DIS
LIN {X -0.132,Y -529.437,Z 347.998,A 0.000,B 0.000,C 90.000,E1 215.678} C_DIS
LIN {X 0.155,Y -524.701,Z 347.989,A 0.000,B 0.000,C 90.000,E1 213.913} C_DIS
LIN {X 0.108,Y -517.470,Z 347.972,A 0.000,B 0.000,C 90.000,E1 211.003} C_DIS
LIN {X 0.082,Y -512.810,Z 347.961,A 0.000,B 0.000,C 90.000,E1 208.949} C_DIS
LIN {X 0.041,Y -508.866,Z 347.951,A 0.000,B 0.000,C 90.000,E1 207.180} C_DIS
LIN {X 0.183,Y -506.306,Z 347.944,A 0.000,B 0.000,C 90.000,E1 205.976} C_DIS
LIN {X -0.084,Y -503.112,Z 347.936,A 0.000,B 0.000,C 90.000,E1 204.515} C_DIS
LIN {X -0.228,Y -500.471,Z 347.930,A 0.000,B 0.000,C 90.000,E1 203.334} C_DIS
LIN {X 0.055,Y -497.759,Z 347.923,A 0.000,B 0.000,C 90.000,E1 202.099} C_DIS
LIN {X -0.113,Y -494.303,Z 347.914,A 0.000,B 0.000,C 90.000,E1 200.610} C_DIS
LIN {X -0.157,Y -489.498,Z 347.903,A 0.000,B 0.000,C 90.000,E1 198.489} C_DIS
LIN {X -0.004,Y -483.689,Z 347.887,A 0.000,B 0.000,C 90.000,E1 195.717} C_DIS
LIN {X 0.047,Y -478.873,Z 347.874,A 0.000,B 0.000,C 90.000,E1 193.244} C_DIS
LIN {X -0.132,Y -475.963,Z 347.865,A 0.000,B 0.000,C 90.000,E1 191.715} C_DIS
LIN {X -0.162,Y -472.545,Z 347.855,A 0.000,B 0.000,C 90.000,E1 189.849} C_DIS
LIN {X 0.212,Y -468.296,Z 347.841,A 0.000,B 0.000,C 90.000,E1 187.296} C_DIS
LIN {X 0.069,Y -464.823,Z 347.828,A 0.000,B 0.000,C 90.000,E1 185.106} C_DIS
LIN {X 0.169,Y -460.286,Z 347.809,A 0.000,B 0.000,C 90.000,E1 181.604} C_DIS
LIN {X 0.143,Y -456.189,Z 347.784,A 0.000,B 0.000,C 90.000,E1 177.135} C_DIS
LIN {X 0.035,Y -454.762,Z 347.768,A 0.000,B 0.000,C 90.000,E1 174.261} C_DIS
LIN {X -0.044,Y -454.246,Z 347.749,A 0.000,B 0.000,C 90.000,E1 170.735} C_DIS
LIN {X 0.090,Y -454.603,Z 347.732,A 0.000,B 0.000,C 90.000,E1 167.825} C_DIS
LIN {X 0.176,Y -456.307,Z 347.713,A 0.000,B 0.000,C 90.000,E1 164.283} C_DIS
LIN {X 0.068,Y -458.059,Z 347.700,A 0.000,B 0.000,C 90.000,E1 162.054} C_DIS
LIN {X -0.033,Y -462.772,Z 347.677,A 0.000,B 0.000,C 90.000,E1 157.922} C_DIS
LIN {X -0.256,Y -468.705,Z 347.656,A 0.000,B 0.000,C 90.000,E1 154.152} C_DIS
LIN {X -0.080,Y -474.365,Z 347.641,A 0.000,B 0.000,C 90.000,E1 151.307} C_DIS
LIN {X -0.080,Y -483.595,Z 347.620,A 0.000,B 0.000,C 90.000,E1 147.582} C_DIS
LIN {X 0.223,Y -492.753,Z 347.603,A 0.000,B 0.000,C 90.000,E1 144.482} C_DIS
LIN {X -0.072,Y -499.578,Z 347.591,A 0.000,B 0.000,C 90.000,E1 142.396} C_DIS
LIN {X 0.139,Y -503.473,Z 347.584,A 0.000,B 0.000,C 90.000,E1 141.170} C_DIS
LIN {X 0.010,Y -507.098,Z 347.578,A 0.000,B 0.000,C 90.000,E1 139.989} C_DIS
LIN {X 0.264,Y -510.579,Z 347.571,A 0.000,B 0.000,C 90.000,E1 138.771} C_DIS
LIN {X -0.310,Y -512.244,Z 347.568,A 0.000,B 0.000,C 90.000,E1 138.243} C_DIS
LIN {X 0.104,Y -514.495,Z 347.563,A 0.000,B 0.000,C 90.000,E1 137.310} C_DIS
LIN {X -0.097,Y -515.812,Z 347.560,A 0.000,B 0.000,C 90.000,E1 136.743} C_DIS
LIN {X 0.000,Y -517.626,Z 347.555,A 0.000,B 0.000,C 90.000,E1 135.850} C_DIS
LIN {X -0.267,Y -519.125,Z 347.550,A 0.000,B 0.000,C 90.000,E1 135.000} C_DIS
LIN {X -0.146,Y -520.265,Z 347.545,A 0.000,B 0.000,C 90.000,E1 134.109} C_DIS
LIN {X -0.014,Y -521.015,Z 347.540,A 0.000,B 0.000,C 90.000,E1 133.218} C_DIS
LIN {X 0.056,Y -521.520,Z 347.534,A 0.000,B 0.000,C 90.000,E1 132.043} C_DIS
LIN {X 0.232,Y -521.558,Z 347.529,A 0.000,B 0.000,C 90.000,E1 131.148} C_DIS
LIN {X 0.016,Y -521.199,Z 347.524,A 0.000,B 0.000,C 90.000,E1 130.297} C_DIS
LIN {X -0.140,Y -520.560,Z 347.519,A 0.000,B 0.000,C 90.000,E1 129.439} C_DIS
LIN {X -0.075,Y -518.848,Z 347.511,A 0.000,B 0.000,C 90.000,E1 127.971} C_DIS
LIN {X -0.113,Y -516.531,Z 347.501,A 0.000,B 0.000,C 90.000,E1 126.217} C_DIS
LIN {X 0.039,Y -514.722,Z 347.495,A 0.000,B 0.000,C 90.000,E1 125.025} C_DIS
LIN {X -0.124,Y -512.782,Z 347.488,A 0.000,B 0.000,C 90.000,E1 123.865} C_DIS
LIN {X -0.031,Y -510.527,Z 347.482,A 0.000,B 0.000,C 90.000,E1 122.673} C_DIS
LIN {X 0.175,Y -508.045,Z 347.475,A 0.000,B 0.000,C 90.000,E1 121.465} C_DIS
LIN {X -0.029,Y -504.790,Z 347.467,A 0.000,B 0.000,C 90.000,E1 120.001} C_DIS
LIN {X -0.161,Y -501.978,Z 347.460,A 0.000,B 0.000,C 90.000,E1 118.821} C_DIS
LIN {X 0.005,Y -497.529,Z 347.450,A 0.000,B 0.000,C 90.000,E1 117.001} C_DIS
LIN {X -0.018,Y -494.374,Z 347.443,A 0.000,B 0.000,C 90.000,E1 115.796} C_DIS
LIN {X -0.084,Y -491.148,Z 347.437,A 0.000,B 0.000,C 90.000,E1 114.591} C_DIS
LIN {X 0.217,Y -488.521,Z 347.432,A 0.000,B 0.000,C 90.000,E1 113.643} C_DIS
LIN {X -0.138,Y -484.890,Z 347.425,A 0.000,B 0.000,C 90.000,E1 112.461} C_DIS
LIN {X -0.096,Y -481.077,Z 347.418,A 0.000,B 0.000,C 90.000,E1 111.227} C_DIS
LIN {X -0.106,Y -477.878,Z 347.413,A 0.000,B 0.000,C 90.000,E1 110.301} C_DIS
LIN {X 0.108,Y -473.489,Z 347.406,A 0.000,B 0.000,C 90.000,E1 109.033} C_DIS
LIN {X -0.191,Y -468.784,Z 347.399,A 0.000,B 0.000,C 90.000,E1 107.819} C_DIS
LIN {X 0.134,Y -464.547,Z 347.393,A 0.000,B 0.000,C 90.000,E1 106.677} C_DIS
LIN {X -0.164,Y -463.855,Z 347.392,A 0.000,B 0.000,C 90.000,E1 106.551} C_DIS
LIN {X 0.240,Y -463.862,Z 347.392,A 0.000,B 0.000,C 90.000,E1 106.496} C_DIS
LIN {X 0.004,Y -467.641,Z 347.383,A 0.000,B 0.000,C 90.000,E1 104.954} C_DIS
LIN {X -0.073,Y -469.565,Z 347.376,A 0.000,B 0.000,C 90.000,E1 103.703} C_DIS
LIN {X -0.038,Y -475.860,Z 347.357,A 0.000,B 0.000,C 90.000,E1 100.254} C_DIS
LIN {X -0.200,Y -476.331,Z 347.355,A 0.000,B 0.000,C 90.000,E1 99.962} C_DIS
LIN {X 0.226,Y -481.833,Z 347.331,A 0.000,B 0.000,C 90.000,E1 95.568} C_DIS
LIN {X 0.073,Y -482.183,Z 347.329,A 0.000,B 0.000,C 90.000,E1 95.277} C_DIS
LIN {X 0.007,Y -485.337,Z 347.305,A 0.000,B 0.000,C 90.000,E1 90.974} C_DIS
LIN {X -0.168,Y -485.534,Z 347.304,A 0.000,B 0.000,C 90.000,E1 90.688} C_DIS
LIN {X 0.039,Y -486.333,Z 347.282,A 0.000,B 0.000,C 90.000,E1 86.674} C_DIS
LIN {X 0.173,Y -486.285,Z 347.278,A 0.000,B 0.000,C 90.000,E1 86.045} C_DIS
LIN {X -0.107,Y -484.694,Z 347.254,A 0.000,B 0.000,C 90.000,E1 81.781} C_DIS
LIN {X -0.238,Y -484.566,Z 347.253,A 0.000,B 0.000,C 90.000,E1 81.489} C_DIS
LIN {X 0.111,Y -480.505,Z 347.227,A 0.000,B 0.000,C 90.000,E1 76.825} C_DIS
LIN {X 0.135,Y -477.002,Z 347.214,A 0.000,B 0.000,C 90.000,E1 74.519} C_DIS
LIN {X 0.095,Y -476.998,Z 347.214,A 0.000,B 0.000,C 90.000,E1 74.519} C_DIS
LIN {X -0.001,Y -480.893,Z 347.210,A 0.000,B 0.000,C 90.000,E1 73.740} C_DIS
LIN {X -0.202,Y -484.925,Z 347.205,A 0.000,B 0.000,C 90.000,E1 72.906} C_DIS
LIN {X -0.105,Y -488.351,Z 347.201,A 0.000,B 0.000,C 90.000,E1 72.127} C_DIS
LIN {X 0.154,Y -490.295,Z 347.198,A 0.000,B 0.000,C 90.000,E1 71.638} C_DIS
LIN {X 0.050,Y -492.671,Z 347.195,A 0.000,B 0.000,C 90.000,E1 71.040} C_DIS
LIN {X 0.050,Y -497.130,Z 347.188,A 0.000,B 0.000,C 90.000,E1 69.826} C_DIS
LIN {X 0.223,Y -500.276,Z 347.183,A 0.000,B 0.000,C 90.000,E1 68.901} C_DIS
LIN {X 0.132,Y -504.937,Z 347.175,A 0.000,B 0.000,C 90.000,E1 67.411} C_DIS
LIN {X -0.067,Y -507.682,Z 347.170,A 0.000,B 0.000,C 90.000,E1 66.538} C_DIS
LIN {X -0.134,Y -511.168,Z 347.163,A 0.000,B 0.000,C 90.000,E1 65.357} C_DIS
LIN {X 0.174,Y -515.413,Z 347.155,A 0.000,B 0.000,C 90.000,E1 63.845} C_DIS
LIN {X -0.036,Y -518.783,Z 347.148,A 0.000,B 0.000,C 90.000,E1 62.692} C_DIS
LIN {X 0.105,Y -523.686,Z 347.139,A 0.000,B 0.000,C 90.000,E1 60.923} C_DIS
LIN {X -0.097,Y -528.631,Z 347.129,A 0.000,B 0.000,C 90.000,E1 59.203} C_DIS
LIN {X 0.080,Y -533.473,Z 347.119,A 0.000,B 0.000,C 90.000,E1 57.454} C_DIS
LIN {X 0.203,Y -537.391,Z 347.111,A 0.000,B 0.000,C 90.000,E1 56.008} C_DIS
LIN {X -0.047,Y -541.024,Z 347.103,A 0.000,B 0.000,C 90.000,E1 54.609} C_DIS
LIN {X 0.024,Y -543.125,Z 347.099,A 0.000,B 0.000,C 90.000,E1 53.749} C_DIS
LIN {X -0.134,Y -546.315,Z 347.091,A 0.000,B 0.000,C 90.000,E1 52.351} C_DIS
LIN {X -0.005,Y -549.139,Z 347.083,A 0.000,B 0.000,C 90.000,E1 50.928} C_DIS
LIN {X -0.222,Y -551.069,Z 347.077,A 0.000,B 0.000,C 90.000,E1 49.828} C_DIS
LIN {X -0.061,Y -552.666,Z 347.071,A 0.000,B 0.000,C 90.000,E1 48.690} C_DIS
LIN {X 0.065,Y -553.577,Z 347.066,A 0.000,B 0.000,C 90.000,E1 47.838} C_DIS
LIN {X -0.149,Y -554.385,Z 347.060,A 0.000,B 0.000,C 90.000,E1 46.743} C_DIS
LIN {X 0.341,Y -554.745,Z 347.057,A 0.000,B 0.000,C 90.000,E1 46.134} C_DIS
LIN {X -0.261,Y -554.786,Z 347.050,A 0.000,B 0.000,C 90.000,E1 45.081} C_DIS
LIN {X 0.269,Y -554.546,Z 347.046,A 0.000,B 0.000,C 90.000,E1 44.190} C_DIS
LIN {X 0.009,Y -554.115,Z 347.041,A 0.000,B 0.000,C 90.000,E1 43.380} C_DIS
LIN {X 0.146,Y -553.524,Z 347.036,A 0.000,B 0.000,C 90.000,E1 42.528} C_DIS
LIN {X -0.078,Y -552.452,Z 347.030,A 0.000,B 0.000,C 90.000,E1 41.434} C_DIS
LIN {X -0.322,Y -551.508,Z 347.026,A 0.000,B 0.000,C 90.000,E1 40.620} C_DIS
LIN {X -0.108,Y -549.828,Z 347.018,A 0.000,B 0.000,C 90.000,E1 39.197} C_DIS
LIN {X -0.322,Y -548.306,Z 347.012,A 0.000,B 0.000,C 90.000,E1 38.096} C_DIS
LIN {X -0.032,Y -546.135,Z 347.002,A 0.000,B 0.000,C 90.000,E1 36.377} C_DIS
LIN {X -0.077,Y -543.633,Z 346.991,A 0.000,B 0.000,C 90.000,E1 34.405} C_DIS
LIN {X -0.041,Y -541.219,Z 346.980,A 0.000,B 0.000,C 90.000,E1 32.418} C_DIS
LIN {X -0.083,Y -539.282,Z 346.971,A 0.000,B 0.000,C 90.000,E1 30.718} C_DIS
LIN {X 0.206,Y -537.146,Z 346.960,A 0.000,B 0.000,C 90.000,E1 28.693} C_DIS
LIN {X 0.279,Y -535.704,Z 346.952,A 0.000,B 0.000,C 90.000,E1 27.257} C_DIS
LIN {X -0.008,Y -533.642,Z 346.941,A 0.000,B 0.000,C 90.000,E1 25.283} C_DIS
LIN {X 0.036,Y -532.586,Z 346.934,A 0.000,B 0.000,C 90.000,E1 24.131} C_DIS
LIN {X -0.277,Y -530.839,Z 346.923,A 0.000,B 0.000,C 90.000,E1 22.153} C_DIS
LIN {X 0.179,Y -529.586,Z 346.913,A 0.000,B 0.000,C 90.000,E1 20.375} C_DIS
LIN {X -0.210,Y -528.081,Z 346.899,A 0.000,B 0.000,C 90.000,E1 17.819} C_DIS
LIN {X -0.145,Y -527.209,Z 346.888,A 0.000,B 0.000,C 90.000,E1 15.788} C_DIS
LIN {X -0.241,Y -526.634,Z 346.876,A 0.000,B 0.000,C 90.000,E1 13.772} C_DIS
LIN {X 0.059,Y -526.434,Z 346.864,A 0.000,B 0.000,C 90.000,E1 11.422} C_DIS
LIN {X 0.215,Y -526.746,Z 346.852,A 0.000,B 0.000,C 90.000,E1 9.378} C_DIS
LIN {X 0.191,Y -527.775,Z 346.836,A 0.000,B 0.000,C 90.000,E1 6.486} C_DIS
LIN {X 0.089,Y -528.888,Z 346.825,A 0.000,B 0.000,C 90.000,E1 4.473} C_DIS
LIN {X -0.076,Y -531.828,Z 346.806,A 0.000,B 0.000,C 90.000,E1 1.031} C_DIS
LIN {X 0.178,Y -534.997,Z 346.791,A 0.000,B 0.000,C 90.000,E1 358.339} C_DIS
LIN {X 0.238,Y -538.345,Z 346.778,A 0.000,B 0.000,C 90.000,E1 356.045} C_DIS
LIN {X -0.185,Y -540.599,Z 346.770,A 0.000,B 0.000,C 90.000,E1 354.666} C_DIS
LIN {X -0.258,Y -545.648,Z 346.755,A 0.000,B 0.000,C 90.000,E1 351.837} C_DIS
LIN {X -0.207,Y -549.911,Z 346.744,A 0.000,B 0.000,C 90.000,E1 349.859} C_DIS
LIN {X -0.169,Y -553.901,Z 346.734,A 0.000,B 0.000,C 90.000,E1 348.173} C_DIS
LIN {X 0.064,Y -560.991,Z 346.720,A 0.000,B 0.000,C 90.000,E1 345.644} C_DIS
LIN {X -0.106,Y -569.329,Z 346.705,A 0.000,B 0.000,C 90.000,E1 342.906} C_DIS
LIN {X -0.175,Y -572.853,Z 346.699,A 0.000,B 0.000,C 90.000,E1 341.819} C_DIS
LIN {X -0.187,Y -578.024,Z 346.690,A 0.000,B 0.000,C 90.000,E1 340.188} C_DIS
LIN {X -0.085,Y -582.371,Z 346.682,A 0.000,B 0.000,C 90.000,E1 338.827} C_DIS
LIN {X 0.176,Y -588.437,Z 346.672,A 0.000,B 0.000,C 90.000,E1 336.922} C_DIS
LIN {X 0.074,Y -596.454,Z 346.659,A 0.000,B 0.000,C 90.000,E1 334.537} C_DIS
LIN {X 0.057,Y -602.837,Z 346.648,A 0.000,B 0.000,C 90.000,E1 332.692} C_DIS
LIN {X -0.023,Y -608.345,Z 346.640,A 0.000,B 0.000,C 90.000,E1 331.129} C_DIS
LIN {X -0.250,Y -614.905,Z 346.630,A 0.000,B 0.000,C 90.000,E1 329.331} C_DIS
LIN {X 0.247,Y -619.574,Z 346.622,A 0.000,B 0.000,C 90.000,E1 327.995} C_DIS
LIN {X 0.296,Y -624.059,Z 346.615,A 0.000,B 0.000,C 90.000,E1 326.707} C_DIS
LIN {X 0.081,Y -626.733,Z 346.611,A 0.000,B 0.000,C 90.000,E1 325.960} C_DIS
LIN {X 0.069,Y -631.737,Z 346.603,A 0.000,B 0.000,C 90.000,E1 324.436} C_DIS
LIN {X 0.014,Y -636.512,Z 346.594,A 0.000,B 0.000,C 90.000,E1 322.924} C_DIS
LIN {X 0.058,Y -641.170,Z 346.586,A 0.000,B 0.000,C 90.000,E1 321.412} C_DIS
LIN {X 0.438,Y -647.533,Z 346.575,A 0.000,B 0.000,C 90.000,E1 319.380} C_DIS
LIN {X 0.238,Y -650.675,Z 346.569,A 0.000,B 0.000,C 90.000,E1 318.405} C_DIS
LIN {X -0.194,Y -659.587,Z 346.554,A 0.000,B 0.000,C 90.000,E1 315.729} C_DIS
LIN {X -0.303,Y -664.233,Z 346.546,A 0.000,B 0.000,C 90.000,E1 314.271} C_DIS
LIN {X 0.156,Y -668.152,Z 346.539,A 0.000,B 0.000,C 90.000,E1 313.014} C_DIS
LIN {X -0.256,Y -672.745,Z 346.531,A 0.000,B 0.000,C 90.000,E1 311.595} C_DIS
LIN {X -0.131,Y -675.511,Z 346.526,A 0.000,B 0.000,C 90.000,E1 310.620} C_DIS
LIN {X -0.350,Y -679.561,Z 346.518,A 0.000,B 0.000,C 90.000,E1 309.197} C_DIS
LIN {X -0.141,Y -682.070,Z 346.512,A 0.000,B 0.000,C 90.000,E1 308.222} C_DIS
LIN {X -0.164,Y -684.914,Z 346.506,A 0.000,B 0.000,C 90.000,E1 307.030} C_DIS
LIN {X -0.307,Y -686.801,Z 346.500,A 0.000,B 0.000,C 90.000,E1 306.091} C_DIS
LIN {X 0.125,Y -688.452,Z 346.495,A 0.000,B 0.000,C 90.000,E1 305.105} C_DIS
LIN {X -0.380,Y -689.747,Z 346.490,A 0.000,B 0.000,C 90.000,E1 304.199} C_DIS
LIN {X -0.149,Y -690.275,Z 346.487,A 0.000,B 0.000,C 90.000,E1 303.706} C_DIS
LIN {X 0.300,Y -690.835,Z 346.483,A 0.000,B 0.000,C 90.000,E1 302.959} C_DIS
LIN {X 0.162,Y -691.124,Z 346.481,A 0.000,B 0.000,C 90.000,E1 302.498} C_DIS
LIN {X 0.397,Y -691.284,Z 346.478,A 0.000,B 0.000,C 90.000,E1 302.005} C_DIS
LIN {X -0.095,Y -691.260,Z 346.474,A 0.000,B 0.000,C 90.000,E1 301.337} C_DIS
LIN {X 0.360,Y -690.876,Z 346.470,A 0.000,B 0.000,C 90.000,E1 300.590} C_DIS
LIN {X 0.228,Y -690.525,Z 346.468,A 0.000,B 0.000,C 90.000,E1 300.129} C_DIS
LIN {X 0.326,Y -689.690,Z 346.464,A 0.000,B 0.000,C 90.000,E1 299.411} C_DIS
LIN {X -0.184,Y -688.670,Z 346.460,A 0.000,B 0.000,C 90.000,E1 298.743} C_DIS
LIN {X 0.275,Y -687.849,Z 346.457,A 0.000,B 0.000,C 90.000,E1 298.231} C_DIS
LIN {X -0.036,Y -686.030,Z 346.452,A 0.000,B 0.000,C 90.000,E1 297.308} C_DIS
LIN {X 0.353,Y -682.932,Z 346.444,A 0.000,B 0.000,C 90.000,E1 295.848} C_DIS
LIN {X 0.281,Y -680.647,Z 346.439,A 0.000,B 0.000,C 90.000,E1 294.899} C_DIS
LIN {X -0.331,Y -677.073,Z 346.431,A 0.000,B 0.000,C 90.000,E1 293.515} C_DIS
LIN {X 0.055,Y -673.898,Z 346.424,A 0.000,B 0.000,C 90.000,E1 292.280} C_DIS
LIN {X -0.165,Y -669.372,Z 346.414,A 0.000,B 0.000,C 90.000,E1 290.610} C_DIS
LIN {X -0.010,Y -665.615,Z 346.406,A 0.000,B 0.000,C 90.000,E1 289.141} C_DIS
LIN {X -0.345,Y -660.794,Z 346.396,A 0.000,B 0.000,C 90.000,E1 287.221} C_DIS
LIN {X -0.277,Y -655.869,Z 346.383,A 0.000,B 0.000,C 90.000,E1 285.009} C_DIS
LIN {X 0.068,Y -651.875,Z 346.372,A 0.000,B 0.000,C 90.000,E1 283.008} C_DIS
LIN {X -0.004,Y -646.706,Z 346.354,A 0.000,B 0.000,C 90.000,E1 279.792} C_DIS
LIN {X 0.292,Y -643.435,Z 346.338,A 0.000,B 0.000,C 90.000,E1 276.777} C_DIS
LIN {X 0.024,Y -641.722,Z 346.324,A 0.000,B 0.000,C 90.000,E1 274.302} C_DIS
LIN {X 0.209,Y -640.667,Z 346.306,A 0.000,B 0.000,C 90.000,E1 271.031} C_DIS
LIN {X 0.326,Y -640.940,Z 346.288,A 0.000,B 0.000,C 90.000,E1 267.764} C_DIS
LIN {X -0.240,Y -641.738,Z 346.277,A 0.000,B 0.000,C 90.000,E1 265.812} C_DIS
LIN {X -0.311,Y -642.502,Z 346.268,A 0.000,B 0.000,C 90.000,E1 264.318} C_DIS
LIN {X -0.089,Y -643.678,Z 346.257,A 0.000,B 0.000,C 90.000,E1 262.299} C_DIS
LIN {X -0.129,Y -644.896,Z 346.248,A 0.000,B 0.000,C 90.000,E1 260.557} C_DIS
LIN {X -0.364,Y -647.252,Z 346.231,A 0.000,B 0.000,C 90.000,E1 257.589} C_DIS
LIN {X 0.199,Y -648.443,Z 346.224,A 0.000,B 0.000,C 90.000,E1 256.297} C_DIS
LIN {X -0.183,Y -649.118,Z 346.219,A 0.000,B 0.000,C 90.000,E1 255.338} C_DIS
LIN {X 0.044,Y -649.396,Z 346.214,A 0.000,B 0.000,C 90.000,E1 254.574} C_DIS
LIN {X -0.178,Y -649.436,Z 346.210,A 0.000,B 0.000,C 90.000,E1 253.850} C_DIS
LIN {X 0.042,Y -649.296,Z 346.206,A 0.000,B 0.000,C 90.000,E1 253.087} C_DIS
LIN {X -0.177,Y -648.884,Z 346.202,A 0.000,B 0.000,C 90.000,E1 252.362} C_DIS
LIN {X 0.073,Y -647.893,Z 346.196,A 0.000,B 0.000,C 90.000,E1 251.348} C_DIS
LIN {X -0.012,Y -647.197,Z 346.194,A 0.000,B 0.000,C 90.000,E1 250.859} C_DIS
LIN {X -0.033,Y -646.056,Z 346.190,A 0.000,B 0.000,C 90.000,E1 250.115} C_DIS
LIN {X -0.122,Y -645.096,Z 346.187,A 0.000,B 0.000,C 90.000,E1 249.625} C_DIS
LIN {X 0.217,Y -643.395,Z 346.183,A 0.000,B 0.000,C 90.000,E1 248.847} C_DIS
LIN {X 0.165,Y -641.410,Z 346.178,A 0.000,B 0.000,C 90.000,E1 248.103} C_DIS
LIN {X 0.097,Y -639.152,Z 346.174,A 0.000,B 0.000,C 90.000,E1 247.358} C_DIS
LIN {X 0.104,Y -635.061,Z 346.167,A 0.000,B 0.000,C 90.000,E1 246.102} C_DIS
LIN {X 0.011,Y -631.657,Z 346.162,A 0.000,B 0.000,C 90.000,E1 245.101} C_DIS
LIN {X 0.139,Y -627.970,Z 346.156,A 0.000,B 0.000,C 90.000,E1 244.076} C_DIS
LIN {X -0.053,Y -623.097,Z 346.149,A 0.000,B 0.000,C 90.000,E1 242.820} C_DIS
LIN {X 0.237,Y -618.301,Z 346.142,A 0.000,B 0.000,C 90.000,E1 241.513} C_DIS
LIN {X -0.089,Y -613.443,Z 346.135,A 0.000,B 0.000,C 90.000,E1 240.255} C_DIS
LIN {X 0.245,Y -606.513,Z 346.125,A 0.000,B 0.000,C 90.000,E1 238.408} C_DIS
LIN {X 0.038,Y -601.576,Z 346.117,A 0.000,B 0.000,C 90.000,E1 237.120} C_DIS
LIN {X -0.357,Y -590.284,Z 346.100,A 0.000,B 0.000,C 90.000,E1 233.989} C_DIS
LIN {X 0.261,Y -587.528,Z 346.095,A 0.000,B 0.000,C 90.000,E1 233.130} C_DIS
LIN {X 0.026,Y -584.566,Z 346.091,A 0.000,B 0.000,C 90.000,E1 232.351} C_DIS
LIN {X 0.213,Y -575.735,Z 346.077,A 0.000,B 0.000,C 90.000,E1 229.908} C_DIS
LIN {X 0.255,Y -569.514,Z 346.067,A 0.000,B 0.000,C 90.000,E1 228.000} C_DIS
LIN {X 0.039,Y -564.048,Z 346.058,A 0.000,B 0.000,C 90.000,E1 226.377} C_DIS
LIN {X -0.306,Y -558.579,Z 346.049,A 0.000,B 0.000,C 90.000,E1 224.757} C_DIS
LIN {X -0.073,Y -554.997,Z 346.042,A 0.000,B 0.000,C 90.000,E1 223.623} C_DIS
LIN {X 0.194,Y -549.652,Z 346.033,A 0.000,B 0.000,C 90.000,E1 221.919} C_DIS
LIN {X -0.014,Y -544.293,Z 346.024,A 0.000,B 0.000,C 90.000,E1 220.253} C_DIS
LIN {X 0.099,Y -538.255,Z 346.013,A 0.000,B 0.000,C 90.000,E1 218.257} C_DIS
LIN {X 0.142,Y -530.699,Z 345.998,A 0.000,B 0.000,C 90.000,E1 215.678} C_DIS
LIN {X -0.275,Y -525.962,Z 345.989,A 0.000,B 0.000,C 90.000,E1 213.992} C_DIS
LIN {X 0.005,Y -518.705,Z 345.973,A 0.000,B 0.000,C 90.000,E1 211.052} C_DIS
LIN {X 0.108,Y -513.416,Z 345.960,A 0.000,B 0.000,C 90.000,E1 208.693} C_DIS
LIN {X -0.181,Y -508.200,Z 345.946,A 0.000,B 0.000,C 90.000,E1 206.360} C_DIS
LIN {X -0.111,Y -504.359,Z 345.936,A 0.000,B 0.000,C 90.000,E1 204.567} C_DIS
LIN {X -0.164,Y -501.092,Z 345.928,A 0.000,B 0.000,C 90.000,E1 203.078} C_DIS
LIN {X 0.057,Y -499.041,Z 345.923,A 0.000,B 0.000,C 90.000,E1 202.153} C_DIS
LIN {X -0.039,Y -494.894,Z 345.913,A 0.000,B 0.000,C 90.000,E1 200.355} C_DIS
LIN {X -0.109,Y -490.817,Z 345.903,A 0.000,B 0.000,C 90.000,E1 198.544} C_DIS
LIN {X -0.050,Y -485.005,Z 345.888,A 0.000,B 0.000,C 90.000,E1 195.788} C_DIS
LIN {X 0.024,Y -479.646,Z 345.872,A 0.000,B 0.000,C 90.000,E1 193.008} C_DIS
LIN {X -0.143,Y -476.733,Z 345.864,A 0.000,B 0.000,C 90.000,E1 191.478} C_DIS
LIN {X 0.005,Y -473.933,Z 345.855,A 0.000,B 0.000,C 90.000,E1 189.905} C_DIS
LIN {X 0.174,Y -469.173,Z 345.839,A 0.000,B 0.000,C 90.000,E1 187.068} C_DIS
LIN {X 0.062,Y -465.706,Z 345.827,A 0.000,B 0.000,C 90.000,E1 184.878} C_DIS
LIN {X -0.224,Y -461.984,Z 345.811,A 0.000,B 0.000,C 90.000,E1 182.064} C_DIS
LIN {X 0.049,Y -459.212,Z 345.797,A 0.000,B 0.000,C 90.000,E1 179.484} C_DIS
LIN {X -0.167,Y -456.369,Z 345.774,A 0.000,B 0.000,C 90.000,E1 175.355} C_DIS
LIN {X 0.193,Y -455.435,Z 345.751,A 0.000,B 0.000,C 90.000,E1 171.141} C_DIS
LIN {X -0.053,Y -455.466,Z 345.742,A 0.000,B 0.000,C 90.000,E1 169.567} C_DIS
LIN {X -0.040,Y -457.169,Z 345.715,A 0.000,B 0.000,C 90.000,E1 164.755} C_DIS
LIN {X -0.009,Y -459.328,Z 345.699,A 0.000,B 0.000,C 90.000,E1 161.873} C_DIS
LIN {X 0.124,Y -464.060,Z 345.676,A 0.000,B 0.000,C 90.000,E1 157.720} C_DIS
LIN {X -0.070,Y -470.619,Z 345.654,A 0.000,B 0.000,C 90.000,E1 153.640} C_DIS
LIN {X -0.012,Y -475.741,Z 345.640,A 0.000,B 0.000,C 90.000,E1 151.129} C_DIS
LIN {X 0.033,Y -485.006,Z 345.619,A 0.000,B 0.000,C 90.000,E1 147.406} C_DIS
LIN {X -0.125,Y -492.267,Z 345.605,A 0.000,B 0.000,C 90.000,E1 144.975} C_DIS
LIN {X 0.229,Y -497.033,Z 345.597,A 0.000,B 0.000,C 90.000,E1 143.417} C_DIS
LIN {X 0.158,Y -502.883,Z 345.587,A 0.000,B 0.000,C 90.000,E1 141.618} C_DIS
LIN {X -0.076,Y -504.785,Z 345.584,A 0.000,B 0.000,C 90.000,E1 141.045} C_DIS
LIN {X 0.035,Y -509.155,Z 345.575,A 0.000,B 0.000,C 90.000,E1 139.542} C_DIS
LIN {X -0.064,Y -512.453,Z 345.569,A 0.000,B 0.000,C 90.000,E1 138.366} C_DIS
LIN {X 0.012,Y -514.702,Z 345.564,A 0.000,B 0.000,C 90.000,E1 137.472} C_DIS
LIN {X 0.080,Y -516.563,Z 345.559,A 0.000,B 0.000,C 90.000,E1 136.581} C_DIS
LIN {X -0.186,Y -518.171,Z 345.554,A 0.000,B 0.000,C 90.000,E1 135.729} C_DIS
LIN {X 0.211,Y -519.832,Z 345.547,A 0.000,B 0.000,C 90.000,E1 134.514} C_DIS
LIN {X -0.019,Y -520.653,Z 345.543,A 0.000,B 0.000,C 90.000,E1 133.662} C_DIS
LIN {X -0.173,Y -521.027,Z 345.539,A 0.000,B 0.000,C 90.000,E1 133.095} C_DIS
LIN {X -0.096,Y -521.368,Z 345.533,A 0.000,B 0.000,C 90.000,E1 131.919} C_DIS
LIN {X 0.084,Y -521.345,Z 345.528,A 0.000,B 0.000,C 90.000,E1 131.024} C_DIS
LIN {X -0.131,Y -520.870,Z 345.523,A 0.000,B 0.000,C 90.000,E1 130.172} C_DIS
LIN {X 0.045,Y -520.008,Z 345.518,A 0.000,B 0.000,C 90.000,E1 129.277} C_DIS
LIN {X 0.036,Y -517.757,Z 345.509,A 0.000,B 0.000,C 90.000,E1 127.523} C_DIS
LIN {X -0.271,Y -515.773,Z 345.500,A 0.000,B 0.000,C 90.000,E1 126.091} C_DIS
LIN {X -0.126,Y -513.946,Z 345.494,A 0.000,B 0.000,C 90.000,E1 124.898} C_DIS
LIN {X 0.070,Y -512.522,Z 345.489,A 0.000,B 0.000,C 90.000,E1 123.992} C_DIS
LIN {X -0.121,Y -510.278,Z 345.482,A 0.000,B 0.000,C 90.000,E1 122.832} C_DIS
LIN {X 0.089,Y -507.814,Z 345.476,A 0.000,B 0.000,C 90.000,E1 121.623} C_DIS
LIN {X 0.142,Y -504.615,Z 345.468,A 0.000,B 0.000,C 90.000,E1 120.129} C_DIS
LIN {X 0.007,Y -501.934,Z 345.461,A 0.000,B 0.000,C 90.000,E1 118.949} C_DIS
LIN {X -0.222,Y -496.829,Z 345.449,A 0.000,B 0.000,C 90.000,E1 116.873} C_DIS
LIN {X 0.145,Y -494.512,Z 345.444,A 0.000,B 0.000,C 90.000,E1 115.924} C_DIS
LIN {X 0.321,Y -490.535,Z 345.436,A 0.000,B 0.000,C 90.000,E1 114.387} C_DIS
LIN {X -0.035,Y -487.916,Z 345.431,A 0.000,B 0.000,C 90.000,E1 113.515} C_DIS
LIN {X 0.051,Y -484.375,Z 345.424,A 0.000,B 0.000,C 90.000,E1 112.280} C_DIS
LIN {X 0.081,Y -481.591,Z 345.419,A 0.000,B 0.000,C 90.000,E1 111.354} C_DIS
LIN {X 0.079,Y -478.665,Z 345.414,A 0.000,B 0.000,C 90.000,E1 110.429} C_DIS
LIN {X -0.168,Y -473.388,Z 345.405,A 0.000,B 0.000,C 90.000,E1 108.906} C_DIS
LIN {X 0.023,Y -470.093,Z 345.400,A 0.000,B 0.000,C 90.000,E1 107.946} C_DIS
LIN {X -0.211,Y -464.333,Z 345.391,A 0.000,B 0.000,C 90.000,E1 106.441} C_DIS
LIN {X -0.005,Y -464.212,Z 345.391,A 0.000,B 0.000,C 90.000,E1 106.386} C_DIS
LIN {X -0.044,Y -464.193,Z 345.391,A 0.000,B 0.000,C 90.000,E1 106.386} C_DIS
LIN {X -0.161,Y -467.551,Z 345.383,A 0.000,B 0.000,C 90.000,E1 105.009} C_DIS
LIN {X 0.023,Y -468.568,Z 345.380,A 0.000,B 0.000,C 90.000,E1 104.356} C_DIS
LIN {X -0.218,Y -475.787,Z 345.357,A 0.000,B 0.000,C 90.000,E1 100.310} C_DIS
LIN {X 0.088,Y -476.299,Z 345.355,A 0.000,B 0.000,C 90.000,E1 99.962} C_DIS
LIN {X 0.036,Y -481.778,Z 345.331,A 0.000,B 0.000,C 90.000,E1 95.625} C_DIS
LIN {X -0.117,Y -482.168,Z 345.330,A 0.000,B 0.000,C 90.000,E1 95.334} C_DIS
LIN {X -0.188,Y -485.301,Z 345.306,A 0.000,B 0.000,C 90.000,E1 91.031} C_DIS
LIN {X 0.122,Y -485.537,Z 345.304,A 0.000,B 0.000,C 90.000,E1 90.688} C_DIS
LIN {X -0.156,Y -486.316,Z 345.282,A 0.000,B 0.000,C 90.000,E1 86.731} C_DIS
LIN {X -0.021,Y -486.309,Z 345.278,A 0.000,B 0.000,C 90.000,E1 86.102} C_DIS
LIN {X 0.183,Y -484.695,Z 345.255,A 0.000,B 0.000,C 90.000,E1 81.781} C_DIS
LIN {X 0.052,Y -484.608,Z 345.253,A 0.000,B 0.000,C 90.000,E1 81.489} C_DIS
LIN {X -0.068,Y -480.540,Z 345.227,A 0.000,B 0.000,C 90.000,E1 76.881} C_DIS
LIN {X -0.174,Y -477.102,Z 345.215,A 0.000,B 0.000,C 90.000,E1 74.629} C_DIS
LIN {X -0.214,Y -477.099,Z 345.215,A 0.000,B 0.000,C 90.000,E1 74.629} C_DIS
LIN {X 0.072,Y -480.354,Z 345.211,A 0.000,B 0.000,C 90.000,E1 73.921} C_DIS
LIN {X -0.099,Y -482.984,Z 345.207,A 0.000,B 0.000,C 90.000,E1 73.323} C_DIS
LIN {X -0.107,Y -484.490,Z 345.206,A 0.000,B 0.000,C 90.000,E1 73.015} C_DIS
LIN {X -0.018,Y -486.420,Z 345.203,A 0.000,B 0.000,C 90.000,E1 72.543} C_DIS
LIN {X -0.010,Y -487.725,Z 345.201,A 0.000,B 0.000,C 90.000,E1 72.236} C_DIS
LIN {X -0.127,Y -490.238,Z 345.198,A 0.000,B 0.000,C 90.000,E1 71.638} C_DIS
LIN {X -0.233,Y -492.573,Z 345.195,A 0.000,B 0.000,C 90.000,E1 71.040} C_DIS
LIN {X -0.187,Y -497.909,Z 345.186,A 0.000,B 0.000,C 90.000,E1 69.518} C_DIS
LIN {X -0.070,Y -499.914,Z 345.183,A 0.000,B 0.000,C 90.000,E1 68.901} C_DIS
LIN {X -0.087,Y -505.383,Z 345.173,A 0.000,B 0.000,C 90.000,E1 67.102} C_DIS
LIN {X -0.090,Y -509.775,Z 345.165,A 0.000,B 0.000,C 90.000,E1 65.613} C_DIS
LIN {X -0.269,Y -514.007,Z 345.156,A 0.000,B 0.000,C 90.000,E1 64.152} C_DIS
LIN {X -0.140,Y -518.215,Z 345.148,A 0.000,B 0.000,C 90.000,E1 62.666} C_DIS
LIN {X -0.308,Y -521.512,Z 345.142,A 0.000,B 0.000,C 90.000,E1 61.513} C_DIS
LIN {X -0.155,Y -527.300,Z 345.130,A 0.000,B 0.000,C 90.000,E1 59.459} C_DIS
LIN {X -0.002,Y -532.185,Z 345.121,A 0.000,B 0.000,C 90.000,E1 57.709} C_DIS
LIN {X 0.250,Y -537.689,Z 345.109,A 0.000,B 0.000,C 90.000,E1 55.674} C_DIS
LIN {X 0.021,Y -541.983,Z 345.100,A 0.000,B 0.000,C 90.000,E1 53.989} C_DIS
LIN {X 0.132,Y -544.663,Z 345.094,A 0.000,B 0.000,C 90.000,E1 52.844} C_DIS
LIN {X -0.147,Y -547.097,Z 345.087,A 0.000,B 0.000,C 90.000,E1 51.743} C_DIS
LIN {X 0.032,Y -549.287,Z 345.081,A 0.000,B 0.000,C 90.000,E1 50.598} C_DIS
LIN {X 0.111,Y -550.755,Z 345.076,A 0.000,B 0.000,C 90.000,E1 49.747} C_DIS
LIN {X -0.094,Y -552.433,Z 345.070,A 0.000,B 0.000,C 90.000,E1 48.647} C_DIS
LIN {X 0.023,Y -553.387,Z 345.066,A 0.000,B 0.000,C 90.000,E1 47.796} C_DIS
LIN {X -0.200,Y -554.303,Z 345.059,A 0.000,B 0.000,C 90.000,E1 46.701} C_DIS
LIN {X 0.322,Y -554.765,Z 345.055,A 0.000,B 0.000,C 90.000,E1 45.810} C_DIS
LIN {X -0.280,Y -554.865,Z 345.049,A 0.000,B 0.000,C 90.000,E1 44.757} C_DIS
LIN {X -0.186,Y -554.740,Z 345.045,A 0.000,B 0.000,C 90.000,E1 44.190} C_DIS
LIN {X -0.041,Y -554.431,Z 345.041,A 0.000,B 0.000,C 90.000,E1 43.338} C_DIS
LIN {X -0.303,Y -553.936,Z 345.036,A 0.000,B 0.000,C 90.000,E1 42.528} C_DIS
LIN {X -0.167,Y -553.275,Z 345.031,A 0.000,B 0.000,C 90.000,E1 41.676} C_DIS
LIN {X 0.019,Y -552.102,Z 345.025,A 0.000,B 0.000,C 90.000,E1 40.539} C_DIS
LIN {X 0.242,Y -550.496,Z 345.017,A 0.000,B 0.000,C 90.000,E1 39.116} C_DIS
LIN {X 0.035,Y -548.984,Z 345.011,A 0.000,B 0.000,C 90.000,E1 38.016} C_DIS
LIN {X 0.334,Y -546.830,Z 345.002,A 0.000,B 0.000,C 90.000,E1 36.297} C_DIS
LIN {X 0.267,Y -544.713,Z 344.992,A 0.000,B 0.000,C 90.000,E1 34.612} C_DIS
LIN {X -0.152,Y -542.621,Z 344.983,A 0.000,B 0.000,C 90.000,E1 32.959} C_DIS
LIN {X -0.161,Y -540.703,Z 344.974,A 0.000,B 0.000,C 90.000,E1 31.258} C_DIS
LIN {X 0.160,Y -538.266,Z 344.961,A 0.000,B 0.000,C 90.000,E1 28.949} C_DIS
LIN {X -0.023,Y -536.521,Z 344.951,A 0.000,B 0.000,C 90.000,E1 27.257} C_DIS
LIN {X 0.140,Y -534.218,Z 344.939,A 0.000,B 0.000,C 90.000,E1 24.951} C_DIS
LIN {X 0.255,Y -533.453,Z 344.934,A 0.000,B 0.000,C 90.000,E1 24.079} C_DIS
LIN {X -0.327,Y -531.469,Z 344.921,A 0.000,B 0.000,C 90.000,E1 21.844} C_DIS
LIN {X 0.143,Y -530.291,Z 344.912,A 0.000,B 0.000,C 90.000,E1 20.066} C_DIS
LIN {X 0.098,Y -529.004,Z 344.899,A 0.000,B 0.000,C 90.000,E1 17.764} C_DIS
LIN {X 0.169,Y -528.278,Z 344.889,A 0.000,B 0.000,C 90.000,E1 16.024} C_DIS
LIN {X 0.123,Y -527.571,Z 344.876,A 0.000,B 0.000,C 90.000,E1 13.716} C_DIS
LIN {X -0.061,Y -527.376,Z 344.863,A 0.000,B 0.000,C 90.000,E1 11.422} C_DIS
LIN {X 0.120,Y -527.698,Z 344.852,A 0.000,B 0.000,C 90.000,E1 9.378} C_DIS
LIN {X 0.092,Y -528.910,Z 344.835,A 0.000,B 0.000,C 90.000,E1 6.201} C_DIS
LIN {X 0.027,Y -530.039,Z 344.823,A 0.000,B 0.000,C 90.000,E1 4.188} C_DIS
LIN {X -0.071,Y -532.787,Z 344.806,A 0.000,B 0.000,C 90.000,E1 1.031} C_DIS
LIN {X 0.196,Y -535.901,Z 344.791,A 0.000,B 0.000,C 90.000,E1 358.339} C_DIS
LIN {X 0.223,Y -537.035,Z 344.786,A 0.000,B 0.000,C 90.000,E1 357.478} C_DIS
LIN {X -0.263,Y -538.779,Z 344.780,A 0.000,B 0.000,C 90.000,E1 356.388} C_DIS
LIN {X -0.136,Y -540.955,Z 344.772,A 0.000,B 0.000,C 90.000,E1 354.951} C_DIS
LIN {X -0.259,Y -545.727,Z 344.756,A 0.000,B 0.000,C 90.000,E1 352.129} C_DIS
LIN {X 0.124,Y -548.770,Z 344.748,A 0.000,B 0.000,C 90.000,E1 350.679} C_DIS
LIN {X -0.049,Y -554.546,Z 344.734,A 0.000,B 0.000,C 90.000,E1 348.173} C_DIS
LIN {X 0.063,Y -560.873,Z 344.722,A 0.000,B 0.000,C 90.000,E1 345.936} C_DIS
LIN {X -0.104,Y -569.087,Z 344.707,A 0.000,B 0.000,C 90.000,E1 343.196} C_DIS
LIN {X 0.003,Y -573.483,Z 344.699,A 0.000,B 0.000,C 90.000,E1 341.819} C_DIS
LIN {X -0.177,Y -577.802,Z 344.691,A 0.000,B 0.000,C 90.000,E1 340.477} C_DIS
LIN {X -0.090,Y -582.991,Z 344.682,A 0.000,B 0.000,C 90.000,E1 338.847} C_DIS
LIN {X -0.142,Y -589.051,Z 344.672,A 0.000,B 0.000,C 90.000,E1 336.975} C_DIS
LIN {X -0.130,Y -596.181,Z 344.660,A 0.000,B 0.000,C 90.000,E1 334.845} C_DIS
LIN {X -0.002,Y -600.697,Z 344.653,A 0.000,B 0.000,C 90.000,E1 333.512} C_DIS
LIN {X -0.279,Y -604.422,Z 344.647,A 0.000,B 0.000,C 90.000,E1 332.487} C_DIS
LIN {X -0.323,Y -609.961,Z 344.638,A 0.000,B 0.000,C 90.000,E1 330.923} C_DIS
LIN {X 0.020,Y -616.583,Z 344.628,A 0.000,B 0.000,C 90.000,E1 329.076} C_DIS
LIN {X 0.017,Y -621.220,Z 344.621,A 0.000,B 0.000,C 90.000,E1 327.788} C_DIS
LIN {X 0.093,Y -625.675,Z 344.614,A 0.000,B 0.000,C 90.000,E1 326.501} C_DIS
LIN {X -0.109,Y -628.218,Z 344.610,A 0.000,B 0.000,C 90.000,E1 325.754} C_DIS
LIN {X 0.276,Y -633.103,Z 344.601,A 0.000,B 0.000,C 90.000,E1 324.196} C_DIS
LIN {X -0.125,Y -637.712,Z 344.593,A 0.000,B 0.000,C 90.000,E1 322.718} C_DIS
LIN {X 0.338,Y -642.181,Z 344.585,A 0.000,B 0.000,C 90.000,E1 321.170} C_DIS
LIN {X -0.010,Y -646.866,Z 344.576,A 0.000,B 0.000,C 90.000,E1 319.703} C_DIS
LIN {X 0.143,Y -650.713,Z 344.569,A 0.000,B 0.000,C 90.000,E1 318.447} C_DIS
LIN {X 0.203,Y -659.495,Z 344.554,A 0.000,B 0.000,C 90.000,E1 315.729} C_DIS
LIN {X 0.107,Y -663.399,Z 344.547,A 0.000,B 0.000,C 90.000,E1 314.514} C_DIS
LIN {X 0.066,Y -667.989,Z 344.539,A 0.000,B 0.000,C 90.000,E1 313.056} C_DIS
LIN {X 0.142,Y -672.527,Z 344.531,A 0.000,B 0.000,C 90.000,E1 311.595} C_DIS
LIN {X 0.284,Y -675.936,Z 344.525,A 0.000,B 0.000,C 90.000,E1 310.378} C_DIS
LIN {X 0.068,Y -679.885,Z 344.517,A 0.000,B 0.000,C 90.000,E1 308.955} C_DIS
LIN {X -0.144,Y -682.296,Z 344.511,A 0.000,B 0.000,C 90.000,E1 308.016} C_DIS
LIN {X 0.253,Y -685.017,Z 344.505,A 0.000,B 0.000,C 90.000,E1 306.790} C_DIS
LIN {X -0.299,Y -686.810,Z 344.499,A 0.000,B 0.000,C 90.000,E1 305.884} C_DIS
LIN {X -0.058,Y -688.039,Z 344.495,A 0.000,B 0.000,C 90.000,E1 305.152} C_DIS
LIN {X -0.006,Y -689.330,Z 344.490,A 0.000,B 0.000,C 90.000,E1 304.199} C_DIS
LIN {X 0.223,Y -689.854,Z 344.487,A 0.000,B 0.000,C 90.000,E1 303.706} C_DIS
LIN {X 0.089,Y -690.385,Z 344.483,A 0.000,B 0.000,C 90.000,E1 303.007} C_DIS
LIN {X -0.055,Y -690.650,Z 344.481,A 0.000,B 0.000,C 90.000,E1 302.546} C_DIS
LIN {X 0.398,Y -690.737,Z 344.477,A 0.000,B 0.000,C 90.000,E1 301.799} C_DIS
LIN {X 0.262,Y -690.646,Z 344.474,A 0.000,B 0.000,C 90.000,E1 301.337} C_DIS
LIN {X -0.003,Y -689.972,Z 344.469,A 0.000,B 0.000,C 90.000,E1 300.413} C_DIS
LIN {X 0.207,Y -689.507,Z 344.466,A 0.000,B 0.000,C 90.000,E1 299.922} C_DIS
LIN {X 0.295,Y -688.550,Z 344.462,A 0.000,B 0.000,C 90.000,E1 299.205} C_DIS
LIN {X 0.376,Y -687.463,Z 344.458,A 0.000,B 0.000,C 90.000,E1 298.487} C_DIS
LIN {X -0.036,Y -685.176,Z 344.452,A 0.000,B 0.000,C 90.000,E1 297.334} C_DIS
LIN {X 0.036,Y -682.039,Z 344.444,A 0.000,B 0.000,C 90.000,E1 295.899} C_DIS
LIN {X -0.137,Y -679.120,Z 344.437,A 0.000,B 0.000,C 90.000,E1 294.719} C_DIS
LIN {X 0.117,Y -675.490,Z 344.429,A 0.000,B 0.000,C 90.000,E1 293.259} C_DIS
LIN {X -0.238,Y -671.562,Z 344.421,A 0.000,B 0.000,C 90.000,E1 291.844} C_DIS
LIN {X 0.155,Y -665.792,Z 344.409,A 0.000,B 0.000,C 90.000,E1 289.631} C_DIS
LIN {X -0.073,Y -660.293,Z 344.397,A 0.000,B 0.000,C 90.000,E1 287.457} C_DIS
LIN {X -0.026,Y -655.323,Z 344.385,A 0.000,B 0.000,C 90.000,E1 285.245} C_DIS
LIN {X 0.049,Y -650.317,Z 344.371,A 0.000,B 0.000,C 90.000,E1 282.771} C_DIS
LIN {X 0.057,Y -645.612,Z 344.354,A 0.000,B 0.000,C 90.000,E1 279.792} C_DIS
LIN {X 0.308,Y -642.341,Z 344.338,A 0.000,B 0.000,C 90.000,E1 276.777} C_DIS
LIN {X 0.005,Y -640.626,Z 344.324,A 0.000,B 0.000,C 90.000,E1 274.302} C_DIS
LIN {X 0.142,Y -639.572,Z 344.306,A 0.000,B 0.000,C 90.000,E1 271.031} C_DIS
LIN {X 0.211,Y -639.850,Z 344.288,A 0.000,B 0.000,C 90.000,E1 267.764} C_DIS
LIN {X 0.010,Y -640.799,Z 344.275,A 0.000,B 0.000,C 90.000,E1 265.527} C_DIS
LIN {X 0.164,Y -641.447,Z 344.268,A 0.000,B 0.000,C 90.000,E1 264.261} C_DIS
LIN {X -0.316,Y -642.158,Z 344.261,A 0.000,B 0.000,C 90.000,E1 263.053} C_DIS
LIN {X -0.025,Y -643.560,Z 344.250,A 0.000,B 0.000,C 90.000,E1 261.027} C_DIS
LIN {X 0.194,Y -644.605,Z 344.242,A 0.000,B 0.000,C 90.000,E1 259.511} C_DIS
LIN {X -0.274,Y -647.009,Z 344.228,A 0.000,B 0.000,C 90.000,E1 257.061} C_DIS
LIN {X -0.051,Y -647.999,Z 344.223,A 0.000,B 0.000,C 90.000,E1 256.047} C_DIS
LIN {X 0.034,Y -648.734,Z 344.217,A 0.000,B 0.000,C 90.000,E1 255.046} C_DIS
LIN {X 0.254,Y -648.990,Z 344.213,A 0.000,B 0.000,C 90.000,E1 254.283} C_DIS
LIN {X -0.110,Y -648.961,Z 344.207,A 0.000,B 0.000,C 90.000,E1 253.323} C_DIS
LIN {X -0.194,Y -648.832,Z 344.205,A 0.000,B 0.000,C 90.000,E1 252.834} C_DIS
LIN {X 0.148,Y -648.607,Z 344.202,A 0.000,B 0.000,C 90.000,E1 252.308} C_DIS
LIN {X -0.016,Y -647.863,Z 344.196,A 0.000,B 0.000,C 90.000,E1 251.329} C_DIS
LIN {X -0.308,Y -647.167,Z 344.194,A 0.000,B 0.000,C 90.000,E1 250.859} C_DIS
LIN {X -0.243,Y -646.952,Z 344.192,A 0.000,B 0.000,C 90.000,E1 250.604} C_DIS
LIN {X 0.279,Y -646.259,Z 344.189,A 0.000,B 0.000,C 90.000,E1 250.061} C_DIS
LIN {X 0.028,Y -644.843,Z 344.185,A 0.000,B 0.000,C 90.000,E1 249.337} C_DIS
LIN {X -0.009,Y -643.180,Z 344.181,A 0.000,B 0.000,C 90.000,E1 248.592} C_DIS
LIN {X -0.058,Y -641.261,Z 344.177,A 0.000,B 0.000,C 90.000,E1 247.847} C_DIS
LIN {X -0.265,Y -637.537,Z 344.170,A 0.000,B 0.000,C 90.000,E1 246.613} C_DIS
LIN {X -0.327,Y -634.245,Z 344.164,A 0.000,B 0.000,C 90.000,E1 245.613} C_DIS
LIN {X -0.167,Y -630.757,Z 344.159,A 0.000,B 0.000,C 90.000,E1 244.588} C_DIS
LIN {X -0.025,Y -626.005,Z 344.152,A 0.000,B 0.000,C 90.000,E1 243.307} C_DIS
LIN {X 0.032,Y -619.307,Z 344.142,A 0.000,B 0.000,C 90.000,E1 241.513} C_DIS
LIN {X 0.259,Y -614.537,Z 344.135,A 0.000,B 0.000,C 90.000,E1 240.205} C_DIS
LIN {X 0.087,Y -607.672,Z 344.125,A 0.000,B 0.000,C 90.000,E1 238.408} C_DIS
LIN {X -0.099,Y -602.797,Z 344.117,A 0.000,B 0.000,C 90.000,E1 237.120} C_DIS
LIN {X 0.385,Y -591.488,Z 344.100,A 0.000,B 0.000,C 90.000,E1 233.909} C_DIS
LIN {X 0.190,Y -588.742,Z 344.095,A 0.000,B 0.000,C 90.000,E1 233.130} C_DIS
LIN {X 0.160,Y -584.764,Z 344.089,A 0.000,B 0.000,C 90.000,E1 232.065} C_DIS
LIN {X -0.091,Y -576.047,Z 344.076,A 0.000,B 0.000,C 90.000,E1 229.666} C_DIS
LIN {X 0.265,Y -570.723,Z 344.067,A 0.000,B 0.000,C 90.000,E1 228.000} C_DIS
LIN {X 0.075,Y -565.284,Z 344.058,A 0.000,B 0.000,C 90.000,E1 226.377} C_DIS
LIN {X -0.245,Y -559.808,Z 344.049,A 0.000,B 0.000,C 90.000,E1 224.757} C_DIS
LIN {X 0.004,Y -556.222,Z 344.042,A 0.000,B 0.000,C 90.000,E1 223.623} C_DIS
LIN {X 0.298,Y -550.874,Z 344.033,A 0.000,B 0.000,C 90.000,E1 221.919} C_DIS
LIN {X 0.114,Y -545.501,Z 344.024,A 0.000,B 0.000,C 90.000,E1 220.253} C_DIS
LIN {X -0.166,Y -539.466,Z 344.013,A 0.000,B 0.000,C 90.000,E1 218.302} C_DIS
LIN {X -0.095,Y -531.906,Z 343.998,A 0.000,B 0.000,C 90.000,E1 215.724} C_DIS
LIN {X -0.057,Y -527.158,Z 343.989,A 0.000,B 0.000,C 90.000,E1 213.992} C_DIS
LIN {X -0.119,Y -520.573,Z 343.974,A 0.000,B 0.000,C 90.000,E1 211.386} C_DIS
LIN {X 0.012,Y -516.506,Z 343.965,A 0.000,B 0.000,C 90.000,E1 209.617} C_DIS
LIN {X 0.057,Y -513.884,Z 343.958,A 0.000,B 0.000,C 90.000,E1 208.437} C_DIS
LIN {X 0.140,Y -509.362,Z 343.947,A 0.000,B 0.000,C 90.000,E1 206.360} C_DIS
LIN {X 0.023,Y -505.523,Z 343.937,A 0.000,B 0.000,C 90.000,E1 204.591} C_DIS
LIN {X 0.199,Y -502.255,Z 343.928,A 0.000,B 0.000,C 90.000,E1 203.078} C_DIS
LIN {X -0.031,Y -500.219,Z 343.923,A 0.000,B 0.000,C 90.000,E1 202.206} C_DIS
LIN {X -0.278,Y -496.106,Z 343.913,A 0.000,B 0.000,C 90.000,E1 200.429} C_DIS
LIN {X -0.117,Y -491.356,Z 343.902,A 0.000,B 0.000,C 90.000,E1 198.290} C_DIS
LIN {X -0.060,Y -486.211,Z 343.888,A 0.000,B 0.000,C 90.000,E1 195.843} C_DIS
LIN {X 0.050,Y -480.875,Z 343.873,A 0.000,B 0.000,C 90.000,E1 193.063} C_DIS
LIN {X 0.223,Y -477.429,Z 343.862,A 0.000,B 0.000,C 90.000,E1 191.186} C_DIS
LIN {X -0.087,Y -474.624,Z 343.854,A 0.000,B 0.000,C 90.000,E1 189.670} C_DIS
LIN {X -0.186,Y -470.427,Z 343.840,A 0.000,B 0.000,C 90.000,E1 187.182} C_DIS
LIN {X -0.003,Y -466.519,Z 343.826,A 0.000,B 0.000,C 90.000,E1 184.645} C_DIS
LIN {X -0.046,Y -463.241,Z 343.812,A 0.000,B 0.000,C 90.000,E1 182.121} C_DIS
LIN {X 0.008,Y -460.181,Z 343.796,A 0.000,B 0.000,C 90.000,E1 179.255} C_DIS
LIN {X -0.125,Y -457.412,Z 343.773,A 0.000,B 0.000,C 90.000,E1 175.122} C_DIS
LIN {X 0.009,Y -456.627,Z 343.748,A 0.000,B 0.000,C 90.000,E1 170.622} C_DIS
LIN {X -0.041,Y -457.666,Z 343.721,A 0.000,B 0.000,C 90.000,E1 165.825} C_DIS
LIN {X 0.213,Y -459.765,Z 343.704,A 0.000,B 0.000,C 90.000,E1 162.598} C_DIS
LIN {X 0.199,Y -464.060,Z 343.681,A 0.000,B 0.000,C 90.000,E1 158.465} C_DIS
LIN {X -0.061,Y -467.135,Z 343.668,A 0.000,B 0.000,C 90.000,E1 156.282} C_DIS
LIN {X -0.149,Y -475.110,Z 343.644,A 0.000,B 0.000,C 90.000,E1 151.897} C_DIS
LIN {X -0.154,Y -484.717,Z 343.621,A 0.000,B 0.000,C 90.000,E1 147.867} C_DIS
LIN {X 0.088,Y -491.808,Z 343.608,A 0.000,B 0.000,C 90.000,E1 145.388} C_DIS
LIN {X 0.006,Y -497.459,Z 343.598,A 0.000,B 0.000,C 90.000,E1 143.577} C_DIS
LIN {X -0.065,Y -503.252,Z 343.588,A 0.000,B 0.000,C 90.000,E1 141.778} C_DIS
LIN {X 0.019,Y -505.154,Z 343.584,A 0.000,B 0.000,C 90.000,E1 141.170} C_DIS
LIN {X 0.141,Y -509.476,Z 343.576,A 0.000,B 0.000,C 90.000,E1 139.666} C_DIS
LIN {X 0.098,Y -512.700,Z 343.569,A 0.000,B 0.000,C 90.000,E1 138.485} C_DIS
LIN {X -0.209,Y -514.909,Z 343.565,A 0.000,B 0.000,C 90.000,E1 137.634} C_DIS
LIN {X -0.141,Y -516.730,Z 343.560,A 0.000,B 0.000,C 90.000,E1 136.743} C_DIS
LIN {X 0.328,Y -518.229,Z 343.555,A 0.000,B 0.000,C 90.000,E1 135.810} C_DIS
LIN {X -0.008,Y -519.797,Z 343.548,A 0.000,B 0.000,C 90.000,E1 134.676} C_DIS
LIN {X 0.121,Y -520.563,Z 343.543,A 0.000,B 0.000,C 90.000,E1 133.785} C_DIS
LIN {X -0.037,Y -520.841,Z 343.540,A 0.000,B 0.000,C 90.000,E1 133.218} C_DIS
LIN {X 0.031,Y -521.155,Z 343.534,A 0.000,B 0.000,C 90.000,E1 132.043} C_DIS
LIN {X -0.086,Y -520.991,Z 343.530,A 0.000,B 0.000,C 90.000,E1 131.472} C_DIS
LIN {X 0.202,Y -521.006,Z 343.529,A 0.000,B 0.000,C 90.000,E1 131.148} C_DIS
LIN {X -0.020,Y -520.501,Z 343.524,A 0.000,B 0.000,C 90.000,E1 130.297} C_DIS
LIN {X 0.147,Y -519.655,Z 343.519,A 0.000,B 0.000,C 90.000,E1 129.402} C_DIS
LIN {X 0.123,Y -517.378,Z 343.509,A 0.000,B 0.000,C 90.000,E1 127.649} C_DIS
LIN {X -0.197,Y -515.396,Z 343.501,A 0.000,B 0.000,C 90.000,E1 126.217} C_DIS
LIN {X -0.061,Y -513.566,Z 343.495,A 0.000,B 0.000,C 90.000,E1 125.025} C_DIS
LIN {X 0.045,Y -511.628,Z 343.488,A 0.000,B 0.000,C 90.000,E1 123.833} C_DIS
LIN {X -0.165,Y -509.371,Z 343.481,A 0.000,B 0.000,C 90.000,E1 122.673} C_DIS
LIN {X -0.084,Y -506.249,Z 343.473,A 0.000,B 0.000,C 90.000,E1 121.180} C_DIS
LIN {X 0.110,Y -503.050,Z 343.465,A 0.000,B 0.000,C 90.000,E1 119.667} C_DIS
LIN {X -0.049,Y -500.262,Z 343.458,A 0.000,B 0.000,C 90.000,E1 118.487} C_DIS
LIN {X 0.072,Y -495.947,Z 343.448,A 0.000,B 0.000,C 90.000,E1 116.668} C_DIS
LIN {X 0.021,Y -492.865,Z 343.442,A 0.000,B 0.000,C 90.000,E1 115.463} C_DIS
LIN {X -0.073,Y -489.772,Z 343.435,A 0.000,B 0.000,C 90.000,E1 114.259} C_DIS
LIN {X 0.035,Y -486.400,Z 343.428,A 0.000,B 0.000,C 90.000,E1 113.025} C_DIS
LIN {X 0.090,Y -483.804,Z 343.423,A 0.000,B 0.000,C 90.000,E1 112.099} C_DIS
LIN {X 0.111,Y -482.025,Z 343.419,A 0.000,B 0.000,C 90.000,E1 111.482} C_DIS
LIN {X 0.114,Y -479.305,Z 343.414,A 0.000,B 0.000,C 90.000,E1 110.556} C_DIS
LIN {X 0.062,Y -475.316,Z 343.407,A 0.000,B 0.000,C 90.000,E1 109.322} C_DIS
LIN {X 0.045,Y -470.088,Z 343.399,A 0.000,B 0.000,C 90.000,E1 107.764} C_DIS
LIN {X -0.109,Y -464.510,Z 343.390,A 0.000,B 0.000,C 90.000,E1 106.260} C_DIS
LIN {X -0.149,Y -464.514,Z 343.390,A 0.000,B 0.000,C 90.000,E1 106.260} C_DIS
LIN {X -0.173,Y -467.694,Z 343.383,A 0.000,B 0.000,C 90.000,E1 104.954} C_DIS
LIN {X -0.216,Y -475.905,Z 343.357,A 0.000,B 0.000,C 90.000,E1 100.254} C_DIS
LIN {X 0.091,Y -476.351,Z 343.355,A 0.000,B 0.000,C 90.000,E1 99.905} C_DIS
LIN {X 0.048,Y -481.868,Z 343.331,A 0.000,B 0.000,C 90.000,E1 95.568} C_DIS
LIN {X -0.104,Y -482.191,Z 343.329,A 0.000,B 0.000,C 90.000,E1 95.277} C_DIS
LIN {X -0.171,Y -485.359,Z 343.305,A 0.000,B 0.000,C 90.000,E1 90.974} C_DIS
LIN {X 0.138,Y -485.532,Z 343.304,A 0.000,B 0.000,C 90.000,E1 90.630} C_DIS
LIN {X -0.139,Y -486.343,Z 343.281,A 0.000,B 0.000,C 90.000,E1 86.674} C_DIS
LIN {X -0.005,Y -486.270,Z 343.278,A 0.000,B 0.000,C 90.000,E1 86.045} C_DIS
LIN {X 0.195,Y -484.693,Z 343.254,A 0.000,B 0.000,C 90.000,E1 81.724} C_DIS
LIN {X 0.063,Y -484.541,Z 343.253,A 0.000,B 0.000,C 90.000,E1 81.432} C_DIS
LIN {X -0.068,Y -480.479,Z 343.227,A 0.000,B 0.000,C 90.000,E1 76.825} C_DIS
LIN {X -0.049,Y -477.198,Z 343.215,A 0.000,B 0.000,C 90.000,E1 74.685} C_DIS
LIN {X -0.090,Y -477.215,Z 343.215,A 0.000,B 0.000,C 90.000,E1 74.685} C_DIS
LIN {X -0.019,Y -480.223,Z 343.211,A 0.000,B 0.000,C 90.000,E1 74.031} C_DIS
LIN {X 0.050,Y -482.244,Z 343.209,A 0.000,B 0.000,C 90.000,E1 73.559} C_DIS
LIN {X 0.070,Y -485.138,Z 343.205,A 0.000,B 0.000,C 90.000,E1 72.851} C_DIS
LIN {X 0.070,Y -486.302,Z 343.203,A 0.000,B 0.000,C 90.000,E1 72.543} C_DIS
LIN {X 0.077,Y -487.624,Z 343.201,A 0.000,B 0.000,C 90.000,E1 72.236} C_DIS
LIN {X -0.060,Y -488.674,Z 343.200,A 0.000,B 0.000,C 90.000,E1 71.945} C_DIS
LIN {X -0.044,Y -489.966,Z 343.198,A 0.000,B 0.000,C 90.000,E1 71.638} C_DIS
LIN {X 0.070,Y -491.558,Z 343.195,A 0.000,B 0.000,C 90.000,E1 71.167} C_DIS
LIN {X -0.116,Y -493.149,Z 343.193,A 0.000,B 0.000,C 90.000,E1 70.732} C_DIS
LIN {X -0.111,Y -497.296,Z 343.186,A 0.000,B 0.000,C 90.000,E1 69.518} C_DIS
LIN {X 0.001,Y -499.289,Z 343.183,A 0.000,B 0.000,C 90.000,E1 68.901} C_DIS
LIN {X -0.030,Y -504.705,Z 343.173,A 0.000,B 0.000,C 90.000,E1 67.102} C_DIS
LIN {X -0.044,Y -509.092,Z 343.165,A 0.000,B 0.000,C 90.000,E1 65.613} C_DIS
LIN {X -0.237,Y -513.320,Z 343.156,A 0.000,B 0.000,C 90.000,E1 64.152} C_DIS
LIN {X -0.121,Y -517.535,Z 343.148,A 0.000,B 0.000,C 90.000,E1 62.666} C_DIS
LIN {X 0.079,Y -521.666,Z 343.140,A 0.000,B 0.000,C 90.000,E1 61.179} C_DIS
LIN {X -0.162,Y -526.649,Z 343.130,A 0.000,B 0.000,C 90.000,E1 59.459} C_DIS
LIN {X -0.023,Y -531.551,Z 343.121,A 0.000,B 0.000,C 90.000,E1 57.709} C_DIS
LIN {X -0.232,Y -536.290,Z 343.111,A 0.000,B 0.000,C 90.000,E1 56.008} C_DIS
LIN {X -0.076,Y -539.279,Z 343.105,A 0.000,B 0.000,C 90.000,E1 54.848} C_DIS
LIN {X -0.008,Y -542.147,Z 343.098,A 0.000,B 0.000,C 90.000,E1 53.703} C_DIS
LIN {X 0.106,Y -544.756,Z 343.092,A 0.000,B 0.000,C 90.000,E1 52.557} C_DIS
LIN {X -0.173,Y -547.167,Z 343.086,A 0.000,B 0.000,C 90.000,E1 51.457} C_DIS
LIN {X 0.003,Y -549.335,Z 343.080,A 0.000,B 0.000,C 90.000,E1 50.312} C_DIS
LIN {X 0.083,Y -550.796,Z 343.075,A 0.000,B 0.000,C 90.000,E1 49.461} C_DIS
LIN {X 0.185,Y -552.054,Z 343.070,A 0.000,B 0.000,C 90.000,E1 48.609} C_DIS
LIN {X -0.067,Y -553.096,Z 343.066,A 0.000,B 0.000,C 90.000,E1 47.796} C_DIS
LIN {X 0.085,Y -554.161,Z 343.059,A 0.000,B 0.000,C 90.000,E1 46.662} C_DIS
LIN {X -0.122,Y -554.842,Z 343.053,A 0.000,B 0.000,C 90.000,E1 45.567} C_DIS
LIN {X 0.063,Y -554.948,Z 343.047,A 0.000,B 0.000,C 90.000,E1 44.433} C_DIS
LIN {X -0.135,Y -554.753,Z 343.041,A 0.000,B 0.000,C 90.000,E1 43.338} C_DIS
LIN {X 0.039,Y -554.171,Z 343.035,A 0.000,B 0.000,C 90.000,E1 42.204} C_DIS
LIN {X -0.190,Y -553.528,Z 343.030,A 0.000,B 0.000,C 90.000,E1 41.391} C_DIS
LIN {X -0.057,Y -552.684,Z 343.025,A 0.000,B 0.000,C 90.000,E1 40.539} C_DIS
LIN {X 0.177,Y -551.109,Z 343.017,A 0.000,B 0.000,C 90.000,E1 39.116} C_DIS
LIN {X 0.032,Y -549.244,Z 343.010,A 0.000,B 0.000,C 90.000,E1 37.729} C_DIS
LIN {X 0.065,Y -546.779,Z 342.999,A 0.000,B 0.000,C 90.000,E1 35.758} C_DIS
LIN {X 0.005,Y -544.686,Z 342.989,A 0.000,B 0.000,C 90.000,E1 34.072} C_DIS
LIN {X 0.091,Y -542.023,Z 342.977,A 0.000,B 0.000,C 90.000,E1 31.799} C_DIS
LIN {X -0.216,Y -540.141,Z 342.967,A 0.000,B 0.000,C 90.000,E1 30.129} C_DIS
LIN {X -0.102,Y -538.423,Z 342.958,A 0.000,B 0.000,C 90.000,E1 28.409} C_DIS
LIN {X -0.054,Y -536.661,Z 342.948,A 0.000,B 0.000,C 90.000,E1 26.693} C_DIS
LIN {X 0.118,Y -534.492,Z 342.936,A 0.000,B 0.000,C 90.000,E1 24.387} C_DIS
LIN {X 0.057,Y -532.690,Z 342.924,A 0.000,B 0.000,C 90.000,E1 22.386} C_DIS
LIN {X 0.054,Y -531.271,Z 342.913,A 0.000,B 0.000,C 90.000,E1 20.375} C_DIS
LIN {X 0.208,Y -529.947,Z 342.900,A 0.000,B 0.000,C 90.000,E1 18.055} C_DIS
LIN {X -0.195,Y -529.083,Z 342.889,A 0.000,B 0.000,C 90.000,E1 16.079} C_DIS
LIN {X -0.071,Y -528.314,Z 342.875,A 0.000,B 0.000,C 90.000,E1 13.467} C_DIS
LIN {X 0.129,Y -528.176,Z 342.864,A 0.000,B 0.000,C 90.000,E1 11.422} C_DIS
LIN {X -0.190,Y -528.500,Z 342.852,A 0.000,B 0.000,C 90.000,E1 9.434} C_DIS
LIN {X -0.155,Y -529.488,Z 342.836,A 0.000,B 0.000,C 90.000,E1 6.543} C_DIS
LIN {X -0.236,Y -530.443,Z 342.827,A 0.000,B 0.000,C 90.000,E1 4.821} C_DIS
LIN {X 0.229,Y -533.183,Z 342.807,A 0.000,B 0.000,C 90.000,E1 1.318} C_DIS
LIN {X 0.208,Y -536.540,Z 342.791,A 0.000,B 0.000,C 90.000,E1 358.339} C_DIS
LIN {X 0.243,Y -537.676,Z 342.786,A 0.000,B 0.000,C 90.000,E1 357.478} C_DIS
LIN {X -0.225,Y -539.823,Z 342.778,A 0.000,B 0.000,C 90.000,E1 356.102} C_DIS
LIN {X -0.084,Y -541.963,Z 342.770,A 0.000,B 0.000,C 90.000,E1 354.666} C_DIS
LIN {X -0.198,Y -546.297,Z 342.756,A 0.000,B 0.000,C 90.000,E1 352.129} C_DIS
LIN {X 0.196,Y -549.337,Z 342.748,A 0.000,B 0.000,C 90.000,E1 350.679} C_DIS
LIN {X 0.041,Y -555.092,Z 342.734,A 0.000,B 0.000,C 90.000,E1 348.173} C_DIS
LIN {X 0.169,Y -561.423,Z 342.722,A 0.000,B 0.000,C 90.000,E1 345.936} C_DIS
LIN {X 0.024,Y -569.620,Z 342.707,A 0.000,B 0.000,C 90.000,E1 343.196} C_DIS
LIN {X 0.142,Y -574.010,Z 342.699,A 0.000,B 0.000,C 90.000,E1 341.819} C_DIS
LIN {X -0.028,Y -578.333,Z 342.692,A 0.000,B 0.000,C 90.000,E1 340.477} C_DIS
LIN {X 0.072,Y -583.507,Z 342.683,A 0.000,B 0.000,C 90.000,E1 338.847} C_DIS
LIN {X 0.151,Y -588.678,Z 342.674,A 0.000,B 0.000,C 90.000,E1 337.230} C_DIS
LIN {X -0.097,Y -593.063,Z 342.666,A 0.000,B 0.000,C 90.000,E1 335.921} C_DIS
LIN {X -0.109,Y -598.524,Z 342.657,A 0.000,B 0.000,C 90.000,E1 334.332} C_DIS
LIN {X -0.069,Y -604.935,Z 342.647,A 0.000,B 0.000,C 90.000,E1 332.487} C_DIS
LIN {X -0.100,Y -610.468,Z 342.638,A 0.000,B 0.000,C 90.000,E1 330.923} C_DIS
LIN {X 0.258,Y -617.084,Z 342.628,A 0.000,B 0.000,C 90.000,E1 329.076} C_DIS
LIN {X 0.265,Y -621.718,Z 342.621,A 0.000,B 0.000,C 90.000,E1 327.788} C_DIS
LIN {X -0.171,Y -626.169,Z 342.614,A 0.000,B 0.000,C 90.000,E1 326.548} C_DIS
LIN {X 0.155,Y -628.709,Z 342.610,A 0.000,B 0.000,C 90.000,E1 325.754} C_DIS
